LIN {X 0,Y 168.066,Z 1160.336,A -85,B 0,C 180,E1 3860.949,E2 3860.949} C_VEL
LIN {X 0,Y 168.839,Z 1157.716,A -85,B 0,C 180,E1 3853.839,E2 3853.839} C_VEL
LIN {X 0,Y 170.872,Z 1154.031,A -85,B 0,C 180,E1 3847.282,E2 3847.282} C_VEL
LIN {X 0,Y 175.431,Z 1147.884,A -85,B 0,C 180,E1 3839.519,E2 3839.519} C_VEL
LIN {X 0,Y 182.099,Z 1140.235,A -85,B 0,C 180,E1 3832.449,E2 3832.449} C_VEL
LIN {X 0,Y 190.542,Z 1131.041,A -85,B 0,C 180,E1 3826.159,E2 3826.159} C_VEL
LIN {X 0,Y 200.886,Z 1120.046,A -85,B 0,C 180,E1 3820.401,E2 3820.401} C_VEL
LIN {X 0,Y 211.702,Z 1108.233,A -85,B 0,C 180,E1 3815.674,E2 3815.674} C_VEL
LIN {X 0,Y 223.761,Z 1094.432,A -85,B 0,C 180,E1 3811.409,E2 3811.409} C_VEL
LIN {X 0,Y 235.465,Z 1080.228,A -85,B 0,C 180,E1 3807.965,E2 3807.965} C_VEL
LIN {X 0,Y 247.528,Z 1064.175,A -85,B 0,C 180,E1 3804.927,E2 3804.927} C_VEL
LIN {X 0,Y 259.432,Z 1046.898,A -85,B 0,C 180,E1 3802.336,E2 3802.336} C_VEL
LIN {X 0,Y 270.34,Z 1029.197,A -85,B 0,C 180,E1 3800.24,E2 3800.24} C_VEL
LIN {X 0,Y 281.272,Z 1009.124,A -85,B 0,C 180,E1 3798.354,E2 3798.354} C_VEL
LIN {X 0,Y 290.529,Z 989.805,A -85,B 0,C 180,E1 3796.914,E2 3796.914} C_VEL
LIN {X 0,Y 299.081,Z 968.565,A -85,B 0,C 180,E1 3795.673,E2 3795.673} C_VEL
LIN {X 0,Y 306.639,Z 946.026,A -85,B 0,C 180,E1 3794.652,E2 3794.652} C_VEL
LIN {X 0,Y 312.105,Z 925.795,A -85,B 0,C 180,E1 3793.953,E2 3793.953} C_VEL
LIN {X 0,Y 316.755,Z 902.819,A -85,B 0,C 180,E1 3793.358,E2 3793.358} C_VEL
LIN {X 0,Y 319.982,Z 878.763,A -85,B 0,C 180,E1 3792.859,E2 3792.859} C_VEL
LIN {X 0,Y 334.332,Z 738.673,A -85,B 0,C 180,E1 3790.249,E2 3790.249} C_VEL
LIN {X 0,Y 331.548,Z 732.932,A -85,B 0,C 180,E1 3787.189,E2 3787.189} C_VEL
LIN {X 0,Y 329.463,Z 728.967,A -85,B 0,C 180,E1 3784.002,E2 3784.002} C_VEL
LIN {X 0,Y 327.825,Z 726.055,A -85,B 0,C 180,E1 3778.951,E2 3778.951} C_VEL
LIN {X 0,Y 327.708,Z 726.631,A -85,B 0,C 180,E1 3776.501,E2 3776.501} C_VEL
LIN {X 0,Y 328.643,Z 729.356,A -85,B 0,C 180,E1 3772.394,E2 3772.394} C_VEL
LIN {X 0,Y 330.208,Z 733.352,A -85,B 0,C 180,E1 3769.356,E2 3769.356} C_VEL
LIN {X 0,Y 332.385,Z 738.672,A -85,B 0,C 180,E1 3766.474,E2 3766.474} C_VEL
LIN {X 0,Y 333.349,Z 741.398,A -85,B 0,C 180,E1 3765.384,E2 3765.384} C_VEL
LIN {X 0,Y 317.82,Z 895.127,A -85,B 0,C 180,E1 3762.622,E2 3762.622} C_VEL
LIN {X 0,Y 313.848,Z 917.711,A -85,B 0,C 180,E1 3762.113,E2 3762.113} C_VEL
LIN {X 0,Y 308.482,Z 939.763,A -85,B 0,C 180,E1 3761.453,E2 3761.453} C_VEL
LIN {X 0,Y 302.074,Z 960.282,A -85,B 0,C 180,E1 3760.622,E2 3760.622} C_VEL
LIN {X 0,Y 294.064,Z 981.25,A -85,B 0,C 180,E1 3759.511,E2 3759.511} C_VEL
LIN {X 0,Y 285.141,Z 1001.061,A -85,B 0,C 180,E1 3758.179,E2 3758.179} C_VEL
LIN {X 0,Y 275.576,Z 1019.159,A -85,B 0,C 180,E1 3756.628,E2 3756.628} C_VEL
LIN {X 0,Y 263.972,Z 1038.466,A -85,B 0,C 180,E1 3754.538,E2 3754.538} C_VEL
LIN {X 0,Y 252.604,Z 1055.305,A -85,B 0,C 180,E1 3752.21,E2 3752.21} C_VEL
LIN {X 0,Y 240.489,Z 1071.192,A -85,B 0,C 180,E1 3749.387,E2 3749.387} C_VEL
LIN {X 0,Y 228.005,Z 1086.134,A -85,B 0,C 180,E1 3745.977,E2 3745.977} C_VEL
LIN {X 0,Y 215.781,Z 1099.645,A -85,B 0,C 180,E1 3741.973,E2 3741.973} C_VEL
LIN {X 0,Y 204.128,Z 1111.522,A -85,B 0,C 180,E1 3737.285,E2 3737.285} C_VEL
LIN {X 0,Y 193.43,Z 1121.957,A -85,B 0,C 180,E1 3731.822,E2 3731.822} C_VEL
LIN {X 0,Y 184.531,Z 1130.557,A -85,B 0,C 180,E1 3725.816,E2 3725.816} C_VEL
LIN {X 0,Y 177.286,Z 1137.575,A -85,B 0,C 180,E1 3719.014,E2 3719.014} C_VEL
LIN {X 0,Y 172.1,Z 1143.09,A -85,B 0,C 180,E1 3711.47,E2 3711.47} C_VEL
LIN {X 0,Y 169.41,Z 1146.62,A -85,B 0,C 180,E1 3704.352,E2 3704.352} C_VEL
LIN {X 0,Y 168.309,Z 1148.543,A -85,B 0,C 180,E1 3697.51,E2 3697.51} C_VEL
LIN {X 0,Y 168.074,Z 1149.252,A -85,B 0,C 180,E1 3691.704,E2 3691.704} C_VEL
LIN {X 0,Y 168.13,Z 1149.097,A -85,B 0,C 180,E1 3685.566,E2 3685.566} C_VEL
LIN {X 0,Y 168.751,Z 1147.654,A -85,B 0,C 180,E1 3678.724,E2 3678.724} C_VEL
LIN {X 0,Y 170.661,Z 1144.912,A -85,B 0,C 180,E1 3671.646,E2 3671.646} C_VEL
LIN {X 0,Y 174.681,Z 1140.291,A -85,B 0,C 180,E1 3664.213,E2 3664.213} C_VEL
LIN {X 0,Y 180.983,Z 1133.995,A -85,B 0,C 180,E1 3657.114,E2 3657.114} C_VEL
LIN {X 0,Y 188.87,Z 1126.429,A -85,B 0,C 180,E1 3650.951,E2 3650.951} C_VEL
LIN {X 0,Y 198.846,Z 1116.798,A -85,B 0,C 180,E1 3645.154,E2 3645.154} C_VEL
LIN {X 0,Y 209.674,Z 1106.072,A -85,B 0,C 180,E1 3640.272,E2 3640.272} C_VEL
LIN {X 0,Y 221.323,Z 1093.753,A -85,B 0,C 180,E1 3636.035,E2 3636.035} C_VEL
LIN {X 0,Y 231.633,Z 1082.102,A -85,B 0,C 180,E1 3632.876,E2 3632.876} C_VEL
LIN {X 0,Y 216.361,Z 1086.384,A -85,B 0,C 180,E1 3628.424,E2 3628.424} C_VEL
LIN {X 0,Y 206.073,Z 1089.051,A -85,B 0,C 180,E1 3624.358,E2 3624.358} C_VEL
LIN {X 0,Y 199.167,Z 1090.87,A -85,B 0,C 180,E1 3620.882,E2 3620.882} C_VEL
LIN {X 0,Y 192.703,Z 1092.575,A -85,B 0,C 180,E1 3616.582,E2 3616.582} C_VEL
LIN {X 0,Y 187.91,Z 1093.996,A -85,B 0,C 180,E1 3612.289,E2 3612.289} C_VEL
LIN {X 0,Y 184.075,Z 1095.335,A -85,B 0,C 180,E1 3607.178,E2 3607.178} C_VEL
LIN {X 0,Y 181.631,Z 1096.889,A -85,B 0,C 180,E1 3600.316,E2 3600.316} C_VEL
LIN {X 0,Y 183.368,Z 1099.077,A -85,B 0,C 180,E1 3589.635,E2 3589.635} C_VEL
LIN {X 0,Y 190.031,Z 1099.894,A -85,B 0,C 180,E1 3581.916,E2 3581.916} C_VEL
LIN {X 0,Y 196.11,Z 1100.057,A -85,B 0,C 180,E1 3577.582,E2 3577.582} C_VEL
LIN {X 0,Y 199.24,Z 1100.523,A -85,B 0,C 180,E1 3575.354,E2 3575.354} C_VEL
LIN {X 0,Y 205.611,Z 1103.158,A -85,B 0,C 180,E1 3570.193,E2 3570.193} C_VEL
LIN {X 0,Y 209.729,Z 1103.302,A -85,B 0,C 180,E1 3568.398,E2 3568.398} C_VEL
LIN {X 0,Y 211.44,Z 1103.162,A -85,B 0,C 180,E1 3567.829,E2 3567.829} C_VEL
LIN {X 0,Y 198.52,Z 1116.738,A -85,B 0,C 180,E1 3562.816,E2 3562.816} C_VEL
LIN {X 0,Y 187.536,Z 1127.926,A -85,B 0,C 180,E1 3557.372,E2 3557.372} C_VEL
LIN {X 0,Y 177.906,Z 1137.495,A -85,B 0,C 180,E1 3551.114,E2 3551.114} C_VEL
LIN {X 0,Y 169.726,Z 1146.03,A -85,B 0,C 180,E1 3543.625,E2 3543.625} C_VEL
LIN {X 0,Y 164.54,Z 1152.122,A -85,B 0,C 180,E1 3536.334,E2 3536.334} C_VEL
LIN {X 0,Y 161.344,Z 1156.757,A -85,B 0,C 180,E1 3528.424,E2 3528.424} C_VEL
LIN {X 0,Y 160.19,Z 1159.484,A -85,B 0,C 180,E1 3521.499,E2 3521.499} C_VEL
LIN {X 0,Y 160.016,Z 1160.978,A -85,B 0,C 180,E1 3514.659,E2 3514.659} C_VEL
LIN {X 0,Y 160.047,Z 1161.226,A -85,B 0,C 180,E1 3508.926,E2 3508.926} C_VEL
LIN {X 0,Y 160.011,Z 1160.594,A -85,B 0,C 180,E1 3503.181,E2 3503.181} C_VEL
LIN {X 0,Y 160.338,Z 1158.972,A -85,B 0,C 180,E1 3497.027,E2 3497.027} C_VEL
LIN {X 0,Y 162.006,Z 1155.698,A -85,B 0,C 180,E1 3489.403,E2 3489.403} C_VEL
LIN {X 0,Y 165.624,Z 1150.678,A -85,B 0,C 180,E1 3481.808,E2 3481.808} C_VEL
LIN {X 0,Y 171.617,Z 1143.989,A -85,B 0,C 180,E1 3474.366,E2 3474.366} C_VEL
LIN {X 0,Y 179.581,Z 1135.749,A -85,B 0,C 180,E1 3467.647,E2 3467.647} C_VEL
LIN {X 0,Y 190.084,Z 1125.198,A -85,B 0,C 180,E1 3461.219,E2 3461.219} C_VEL
LIN {X 0,Y 201.378,Z 1113.79,A -85,B 0,C 180,E1 3455.971,E2 3455.971} C_VEL
LIN {X 0,Y 213.404,Z 1100.89,A -85,B 0,C 180,E1 3451.491,E2 3451.491} C_VEL
LIN {X 0,Y 226.562,Z 1085.934,A -85,B 0,C 180,E1 3447.495,E2 3447.495} C_VEL
LIN {X 0,Y 239.155,Z 1070.454,A -85,B 0,C 180,E1 3444.298,E2 3444.298} C_VEL
LIN {X 0,Y 251.201,Z 1054.032,A -85,B 0,C 180,E1 3441.657,E2 3441.657} C_VEL
LIN {X 0,Y 262.913,Z 1036.48,A -85,B 0,C 180,E1 3439.412,E2 3439.412} C_VEL
LIN {X 0,Y 273.298,Z 1018.853,A -85,B 0,C 180,E1 3437.628,E2 3437.628} C_VEL
LIN {X 0,Y 283.934,Z 998.39,A -85,B 0,C 180,E1 3435.98,E2 3435.98} C_VEL
LIN {X 0,Y 292.6,Z 979.055,A -85,B 0,C 180,E1 3434.748,E2 3434.748} C_VEL
LIN {X 0,Y 300.502,Z 958.071,A -85,B 0,C 180,E1 3433.694,E2 3433.694} C_VEL
LIN {X 0,Y 307.329,Z 936.133,A -85,B 0,C 180,E1 3432.838,E2 3432.838} C_VEL
LIN {X 0,Y 312.656,Z 913.731,A -85,B 0,C 180,E1 3432.199,E2 3432.199} C_VEL
LIN {X 0,Y 316.677,Z 889.714,A -85,B 0,C 180,E1 3431.675,E2 3431.675} C_VEL
LIN {X 0,Y 332.049,Z 744.44,A -85,B 0,C 180,E1 3429.008,E2 3429.008} C_VEL
LIN {X 0,Y 329.883,Z 739.96,A -85,B 0,C 180,E1 3426.351,E2 3426.351} C_VEL
LIN {X 0,Y 328.38,Z 736.839,A -85,B 0,C 180,E1 3423.84,E2 3423.84} C_VEL
LIN {X 0,Y 326.831,Z 733.964,A -85,B 0,C 180,E1 3418.772,E2 3418.772} C_VEL
LIN {X 0,Y 326.748,Z 734.814,A -85,B 0,C 180,E1 3416.139,E2 3416.139} C_VEL
LIN {X 0,Y 327.589,Z 737.286,A -85,B 0,C 180,E1 3412.546,E2 3412.546} C_VEL
LIN {X 0,Y 329.057,Z 741.202,A -85,B 0,C 180,E1 3409.584,E2 3409.584} C_VEL
LIN {X 0,Y 331.095,Z 746.453,A -85,B 0,C 180,E1 3406.776,E2 3406.776} C_VEL
LIN {X 0,Y 331.165,Z 747.084,A -85,B 0,C 180,E1 3406.642,E2 3406.642} C_VEL
LIN {X 0,Y 315.809,Z 895.146,A -85,B 0,C 180,E1 3404.026,E2 3404.026} C_VEL
LIN {X 0,Y 311.75,Z 917.772,A -85,B 0,C 180,E1 3403.53,E2 3403.53} C_VEL
LIN {X 0,Y 306.264,Z 939.882,A -85,B 0,C 180,E1 3402.891,E2 3402.891} C_VEL
LIN {X 0,Y 299.957,Z 959.745,A -85,B 0,C 180,E1 3402.115,E2 3402.115} C_VEL
LIN {X 0,Y 291.791,Z 980.838,A -85,B 0,C 180,E1 3401.041,E2 3401.041} C_VEL
LIN {X 0,Y 282.894,Z 1000.319,A -85,B 0,C 180,E1 3399.782,E2 3399.782} C_VEL
LIN {X 0,Y 272.487,Z 1019.611,A -85,B 0,C 180,E1 3398.18,E2 3398.18} C_VEL
LIN {X 0,Y 260.713,Z 1038.7,A -85,B 0,C 180,E1 3396.159,E2 3396.159} C_VEL
LIN {X 0,Y 248.93,Z 1055.677,A -85,B 0,C 180,E1 3393.86,E2 3393.86} C_VEL
LIN {X 0,Y 236.455,Z 1071.542,A -85,B 0,C 180,E1 3391.082,E2 3391.082} C_VEL
LIN {X 0,Y 223.549,Z 1086.464,A -85,B 0,C 180,E1 3387.708,E2 3387.708} C_VEL
LIN {X 0,Y 211.489,Z 1099.298,A -85,B 0,C 180,E1 3383.944,E2 3383.944} C_VEL
LIN {X 0,Y 199.818,Z 1110.717,A -85,B 0,C 180,E1 3379.516,E2 3379.516} C_VEL
LIN {X 0,Y 188.909,Z 1120.93,A -85,B 0,C 180,E1 3374.319,E2 3374.319} C_VEL
LIN {X 0,Y 179.601,Z 1129.317,A -85,B 0,C 180,E1 3368.574,E2 3368.574} C_VEL
LIN {X 0,Y 171.32,Z 1136.805,A -85,B 0,C 180,E1 3361.559,E2 3361.559} C_VEL
LIN {X 0,Y 165.538,Z 1142.429,A -85,B 0,C 180,E1 3354.208,E2 3354.208} C_VEL
LIN {X 0,Y 162.098,Z 1146.161,A -85,B 0,C 180,E1 3346.852,E2 3346.852} C_VEL
LIN {X 0,Y 160.483,Z 1148.584,A -85,B 0,C 180,E1 3339.322,E2 3339.322} C_VEL
LIN {X 0,Y 160.089,Z 1149.48,A -85,B 0,C 180,E1 3332.864,E2 3332.864} C_VEL
LIN {X 0,Y 160.085,Z 1149.51,A -85,B 0,C 180,E1 3327.494,E2 3327.494} C_VEL
LIN {X 0,Y 160.396,Z 1148.736,A -85,B 0,C 180,E1 3321.396,E2 3321.396} C_VEL
LIN {X 0,Y 161.958,Z 1146.373,A -85,B 0,C 180,E1 3313.502,E2 3313.502} C_VEL
LIN {X 0,Y 165.444,Z 1142.551,A -85,B 0,C 180,E1 3305.865,E2 3305.865} C_VEL
LIN {X 0,Y 171.142,Z 1137.021,A -85,B 0,C 180,E1 3298.538,E2 3298.538} C_VEL
LIN {X 0,Y 179.099,Z 1129.86,A -85,B 0,C 180,E1 3291.707,E2 3291.707} C_VEL
LIN {X 0,Y 188.81,Z 1121.095,A -85,B 0,C 180,E1 3285.651,E2 3285.651} C_VEL
LIN {X 0,Y 199.71,Z 1110.923,A -85,B 0,C 180,E1 3280.448,E2 3280.448} C_VEL
LIN {X 0,Y 211.376,Z 1099.547,A -85,B 0,C 180,E1 3276.014,E2 3276.014} C_VEL
LIN {X 0,Y 221.91,Z 1088.357,A -85,B 0,C 180,E1 3272.654,E2 3272.654} C_VEL
LIN {X 0,Y 211.435,Z 1091.167,A -85,B 0,C 180,E1 3269.527,E2 3269.527} C_VEL
LIN {X 0,Y 201.236,Z 1093.692,A -85,B 0,C 180,E1 3265.612,E2 3265.612} C_VEL
LIN {X 0,Y 193.118,Z 1095.612,A -85,B 0,C 180,E1 3261.568,E2 3261.568} C_VEL
LIN {X 0,Y 187.13,Z 1097.099,A -85,B 0,C 180,E1 3257.732,E2 3257.732} C_VEL
LIN {X 0,Y 181.506,Z 1098.586,A -85,B 0,C 180,E1 3252.73,E2 3252.73} C_VEL
LIN {X 0,Y 177.713,Z 1099.879,A -85,B 0,C 180,E1 3247.761,E2 3247.761} C_VEL
LIN {X 0,Y 175.075,Z 1101.482,A -85,B 0,C 180,E1 3240.328,E2 3240.328} C_VEL
LIN {X 0,Y 176.758,Z 1103.63,A -85,B 0,C 180,E1 3229.572,E2 3229.572} C_VEL
LIN {X 0,Y 183.457,Z 1104.491,A -85,B 0,C 180,E1 3221.573,E2 3221.573} C_VEL
LIN {X 0,Y 191.592,Z 1104.607,A -85,B 0,C 180,E1 3215.981,E2 3215.981} C_VEL
LIN {X 0,Y 203.409,Z 1103.964,A -85,B 0,C 180,E1 3210.558,E2 3210.558} C_VEL
LIN {X 0,Y 209.729,Z 1103.302,A -85,B 0,C 180,E1 3208.398,E2 3208.398} C_VEL
LIN {X 0,Y 210.064,Z 1103.848,A -85,B 0,C 180,E1 3207.907,E2 3207.907} C_VEL
LIN {X 0,Y 208.692,Z 1105.572,A -85,B 0,C 180,E1 3207.279,E2 3207.279} C_VEL
LIN {X 0,Y 205.22,Z 1108.258,A -85,B 0,C 180,E1 3206.659,E2 3206.659} C_VEL
LIN {X 0,Y 196.789,Z 1113.88,A -85,B 0,C 180,E1 3205.674,E2 3205.674} C_VEL
LIN {X 0,Y 193.755,Z 1116.236,A -85,B 0,C 180,E1 3204.876,E2 3204.876} C_VEL
LIN {X 0,Y 181.945,Z 1127.613,A -85,B 0,C 180,E1 3199.321,E2 3199.321} C_VEL
LIN {X 0,Y 171.674,Z 1137.184,A -85,B 0,C 180,E1 3192.956,E2 3192.956} C_VEL
LIN {X 0,Y 162.826,Z 1145.732,A -85,B 0,C 180,E1 3185.246,E2 3185.246} C_VEL
LIN {X 0,Y 157.136,Z 1151.819,A -85,B 0,C 180,E1 3177.678,E2 3177.678} C_VEL
LIN {X 0,Y 153.574,Z 1156.459,A -85,B 0,C 180,E1 3169.393,E2 3169.393} C_VEL
LIN {X 0,Y 152.246,Z 1159.182,A -85,B 0,C 180,E1 3162.132,E2 3162.132} C_VEL
LIN {X 0,Y 152.013,Z 1160.659,A -85,B 0,C 180,E1 3155.284,E2 3155.284} C_VEL
LIN {X 0,Y 152.05,Z 1160.959,A -85,B 0,C 180,E1 3149.247,E2 3149.247} C_VEL
LIN {X 0,Y 152.014,Z 1160.375,A -85,B 0,C 180,E1 3143.201,E2 3143.201} C_VEL
LIN {X 0,Y 152.366,Z 1158.799,A -85,B 0,C 180,E1 3136.722,E2 3136.722} C_VEL
LIN {X 0,Y 154.054,Z 1155.753,A -85,B 0,C 180,E1 3129.086,E2 3129.086} C_VEL
LIN {X 0,Y 158.043,Z 1150.711,A -85,B 0,C 180,E1 3120.847,E2 3120.847} C_VEL
LIN {X 0,Y 164.538,Z 1144.048,A -85,B 0,C 180,E1 3113.015,E2 3113.015} C_VEL
LIN {X 0,Y 173.013,Z 1135.859,A -85,B 0,C 180,E1 3106.093,E2 3106.093} C_VEL
LIN {X 0,Y 184.457,Z 1125.072,A -85,B 0,C 180,E1 3099.36,E2 3099.36} C_VEL
LIN {X 0,Y 196.558,Z 1113.462,A -85,B 0,C 180,E1 3093.988,E2 3093.988} C_VEL
LIN {X 0,Y 209.352,Z 1100.343,A -85,B 0,C 180,E1 3089.466,E2 3089.466} C_VEL
LIN {X 0,Y 223.373,Z 1084.955,A -85,B 0,C 180,E1 3085.449,E2 3085.449} C_VEL
LIN {X 0,Y 236.638,Z 1069.116,A -85,B 0,C 180,E1 3082.281,E2 3082.281} C_VEL
LIN {X 0,Y 249.192,Z 1052.348,A -85,B 0,C 180,E1 3079.696,E2 3079.696} C_VEL
LIN {X 0,Y 261.961,Z 1033.33,A -85,B 0,C 180,E1 3077.406,E2 3077.406} C_VEL
LIN {X 0,Y 273.075,Z 1014.66,A -85,B 0,C 180,E1 3075.641,E2 3075.641} C_VEL
LIN {X 0,Y 283.102,Z 995.111,A -85,B 0,C 180,E1 3074.192,E2 3074.192} C_VEL
LIN {X 0,Y 291.964,Z 975.24,A -85,B 0,C 180,E1 3073.018,E2 3073.018} C_VEL
LIN {X 0,Y 299.128,Z 956.022,A -85,B 0,C 180,E1 3072.12,E2 3072.12} C_VEL
LIN {X 0,Y 306.111,Z 933.229,A -85,B 0,C 180,E1 3071.294,E2 3071.294} C_VEL
LIN {X 0,Y 311.322,Z 911.208,A -85,B 0,C 180,E1 3070.707,E2 3070.707} C_VEL
LIN {X 0,Y 315.043,Z 888.222,A -85,B 0,C 180,E1 3070.228,E2 3070.228} C_VEL
LIN {X 0,Y 329.913,Z 750.378,A -85,B 0,C 180,E1 3067.75,E2 3067.75} C_VEL
LIN {X 0,Y 328.35,Z 747.083,A -85,B 0,C 180,E1 3065.591,E2 3065.591} C_VEL
LIN {X 0,Y 327.21,Z 744.588,A -85,B 0,C 180,E1 3063.503,E2 3063.503} C_VEL
LIN {X 0,Y 325.856,Z 741.909,A -85,B 0,C 180,E1 3058.769,E2 3058.769} C_VEL
LIN {X 0,Y 325.759,Z 742.699,A -85,B 0,C 180,E1 3056.304,E2 3056.304} C_VEL
LIN {X 0,Y 326.514,Z 745.1,A -85,B 0,C 180,E1 3052.787,E2 3052.787} C_VEL
LIN {X 0,Y 327.861,Z 748.907,A -85,B 0,C 180,E1 3049.9,E2 3049.9} C_VEL
LIN {X 0,Y 329.155,Z 752.529,A -85,B 0,C 180,E1 3047.92,E2 3047.92} C_VEL
LIN {X 0,Y 314.011,Z 894.992,A -85,B 0,C 180,E1 3045.451,E2 3045.451} C_VEL
LIN {X 0,Y 309.874,Z 917.703,A -85,B 0,C 180,E1 3044.969,E2 3044.969} C_VEL
LIN {X 0,Y 304.241,Z 940,A -85,B 0,C 180,E1 3044.349,E2 3044.349} C_VEL
LIN {X 0,Y 297.606,Z 960.483,A -85,B 0,C 180,E1 3043.575,E2 3043.575} C_VEL
LIN {X 0,Y 289.293,Z 981.419,A -85,B 0,C 180,E1 3042.539,E2 3042.539} C_VEL
LIN {X 0,Y 280.225,Z 1000.82,A -85,B 0,C 180,E1 3041.32,E2 3041.32} C_VEL
LIN {X 0,Y 270.066,Z 1019.262,A -85,B 0,C 180,E1 3039.837,E2 3039.837} C_VEL
LIN {X 0,Y 257.968,Z 1038.499,A -85,B 0,C 180,E1 3037.872,E2 3037.872} C_VEL
LIN {X 0,Y 245.867,Z 1055.521,A -85,B 0,C 180,E1 3035.635,E2 3035.635} C_VEL
LIN {X 0,Y 233.245,Z 1071.161,A -85,B 0,C 180,E1 3032.973,E2 3032.973} C_VEL
LIN {X 0,Y 220.026,Z 1086.037,A -85,B 0,C 180,E1 3029.702,E2 3029.702} C_VEL
LIN {X 0,Y 207.46,Z 1098.936,A -85,B 0,C 180,E1 3025.992,E2 3025.992} C_VEL
LIN {X 0,Y 195.214,Z 1110.471,A -85,B 0,C 180,E1 3021.596,E2 3021.596} C_VEL
LIN {X 0,Y 183.676,Z 1120.789,A -85,B 0,C 180,E1 3016.386,E2 3016.386} C_VEL
LIN {X 0,Y 173.268,Z 1129.62,A -85,B 0,C 180,E1 3010.264,E2 3010.264} C_VEL
LIN {X 0,Y 164.511,Z 1137.013,A -85,B 0,C 180,E1 3003.161,E2 3003.161} C_VEL
LIN {X 0,Y 158.158,Z 1142.704,A -85,B 0,C 180,E1 2995.461,E2 2995.461} C_VEL
LIN {X 0,Y 154.349,Z 1146.456,A -85,B 0,C 180,E1 2987.726,E2 2987.726} C_VEL
LIN {X 0,Y 152.548,Z 1148.877,A -85,B 0,C 180,E1 2979.812,E2 2979.812} C_VEL
LIN {X 0,Y 152.097,Z 1149.771,A -85,B 0,C 180,E1 2973.015,E2 2973.015} C_VEL
LIN {X 0,Y 152.091,Z 1149.801,A -85,B 0,C 180,E1 2967.362,E2 2967.362} C_VEL
LIN {X 0,Y 152.443,Z 1149.028,A -85,B 0,C 180,E1 2960.943,E2 2960.943} C_VEL
LIN {X 0,Y 154.196,Z 1146.668,A -85,B 0,C 180,E1 2952.646,E2 2952.646} C_VEL
LIN {X 0,Y 157.881,Z 1142.976,A -85,B 0,C 180,E1 2944.893,E2 2944.893} C_VEL
LIN {X 0,Y 164.098,Z 1137.416,A -85,B 0,C 180,E1 2937.161,E2 2937.161} C_VEL
LIN {X 0,Y 172.737,Z 1130.161,A -85,B 0,C 180,E1 2930.021,E2 2930.021} C_VEL
LIN {X 0,Y 182.708,Z 1121.67,A -85,B 0,C 180,E1 2924.028,E2 2924.028} C_VEL
LIN {X 0,Y 194.497,Z 1111.231,A -85,B 0,C 180,E1 2918.611,E2 2918.611} C_VEL
LIN {X 0,Y 206.99,Z 1099.549,A -85,B 0,C 180,E1 2914.08,E2 2914.08} C_VEL
LIN {X 0,Y 211.969,Z 1094.464,A -85,B 0,C 180,E1 2912.45,E2 2912.45} C_VEL
LIN {X 0,Y 196.359,Z 1098.097,A -85,B 0,C 180,E1 2906.949,E2 2906.949} C_VEL
LIN {X 0,Y 183.195,Z 1101.206,A -85,B 0,C 180,E1 2900.112,E2 2900.112} C_VEL
LIN {X 0,Y 171.637,Z 1104.182,A -85,B 0,C 180,E1 2889.05,E2 2889.05} C_VEL
LIN {X 0,Y 169.799,Z 1107.852,A -85,B 0,C 180,E1 2869.826,E2 2869.826} C_VEL
LIN {X 0,Y 176.708,Z 1108.791,A -85,B 0,C 180,E1 2861.186,E2 2861.186} C_VEL
LIN {X 0,Y 185.45,Z 1108.965,A -85,B 0,C 180,E1 2855.132,E2 2855.132} C_VEL
LIN {X 0,Y 197.588,Z 1108.421,A -85,B 0,C 180,E1 2849.601,E2 2849.601} C_VEL
LIN {X 0,Y 202.008,Z 1108.039,A -85,B 0,C 180,E1 2848.064,E2 2848.064} C_VEL
LIN {X 0,Y 193.755,Z 1116.236,A -85,B 0,C 180,E1 2844.876,E2 2844.876} C_VEL
LIN {X 0,Y 189.106,Z 1120.152,A -85,B 0,C 180,E1 2843.4,E2 2843.4} C_VEL
LIN {X 0,Y 174.971,Z 1129.302,A -85,B 0,C 180,E1 2839.934,E2 2839.934} C_VEL
LIN {X 0,Y 170.613,Z 1132.534,A -85,B 0,C 180,E1 2838.109,E2 2838.109} C_VEL
LIN {X 0,Y 160.546,Z 1141.375,A -85,B 0,C 180,E1 2831.101,E2 2831.101} C_VEL
LIN {X 0,Y 152.816,Z 1148.567,A -85,B 0,C 180,E1 2823.34,E2 2823.34} C_VEL
LIN {X 0,Y 147.706,Z 1153.814,A -85,B 0,C 180,E1 2815.244,E2 2815.244} C_VEL
LIN {X 0,Y 144.832,Z 1157.781,A -85,B 0,C 180,E1 2806.442,E2 2806.442} C_VEL
LIN {X 0,Y 144.065,Z 1159.796,A -85,B 0,C 180,E1 2798.783,E2 2798.783} C_VEL
LIN {X 0,Y 144.036,Z 1160.549,A -85,B 0,C 180,E1 2792.785,E2 2792.785} C_VEL
LIN {X 0,Y 144.043,Z 1160.571,A -85,B 0,C 180,E1 2787.613,E2 2787.613} C_VEL
LIN {X 0,Y 144.049,Z 1159.86,A -85,B 0,C 180,E1 2781.619,E2 2781.619} C_VEL
LIN {X 0,Y 144.685,Z 1158.011,A -85,B 0,C 180,E1 2774.365,E2 2774.365} C_VEL
LIN {X 0,Y 147.338,Z 1154.222,A -85,B 0,C 180,E1 2765.546,E2 2765.546} C_VEL
LIN {X 0,Y 152.222,Z 1149.065,A -85,B 0,C 180,E1 2757.411,E2 2757.411} C_VEL
LIN {X 0,Y 159.901,Z 1141.895,A -85,B 0,C 180,E1 2749.435,E2 2749.435} C_VEL
LIN {X 0,Y 169.566,Z 1133.424,A -85,B 0,C 180,E1 2742.517,E2 2742.517} C_VEL
LIN {X 0,Y 181.247,Z 1122.963,A -85,B 0,C 180,E1 2736.349,E2 2736.349} C_VEL
LIN {X 0,Y 194.798,Z 1110.385,A -85,B 0,C 180,E1 2730.881,E2 2730.881} C_VEL
LIN {X 0,Y 208.068,Z 1097.345,A -85,B 0,C 180,E1 2726.643,E2 2726.643} C_VEL
LIN {X 0,Y 221.674,Z 1082.643,A -85,B 0,C 180,E1 2723.053,E2 2723.053} C_VEL
LIN {X 0,Y 236.039,Z 1065.64,A -85,B 0,C 180,E1 2719.882,E2 2719.882} C_VEL
LIN {X 0,Y 248.926,Z 1048.73,A -85,B 0,C 180,E1 2717.452,E2 2717.452} C_VEL
LIN {X 0,Y 260.999,Z 1030.713,A -85,B 0,C 180,E1 2715.445,E2 2715.445} C_VEL
LIN {X 0,Y 272.733,Z 1010.921,A -85,B 0,C 180,E1 2713.708,E2 2713.708} C_VEL
LIN {X 0,Y 282.549,Z 991.834,A -85,B 0,C 180,E1 2712.396,E2 2712.396} C_VEL
LIN {X 0,Y 291.658,Z 970.97,A -85,B 0,C 180,E1 2711.268,E2 2711.268} C_VEL
LIN {X 0,Y 299.269,Z 950.317,A -85,B 0,C 180,E1 2710.393,E2 2710.393} C_VEL
LIN {X 0,Y 305.458,Z 929.062,A -85,B 0,C 180,E1 2709.708,E2 2709.708} C_VEL
LIN {X 0,Y 310.715,Z 905.521,A -85,B 0,C 180,E1 2709.14,E2 2709.14} C_VEL
LIN {X 0,Y 314.102,Z 882.99,A -85,B 0,C 180,E1 2708.699,E2 2708.699} C_VEL
LIN {X 0,Y 327.933,Z 756.407,A -85,B 0,C 180,E1 2706.477,E2 2706.477} C_VEL
LIN {X 0,Y 326.135,Z 752.46,A -85,B 0,C 180,E1 2703.339,E2 2703.339} C_VEL
LIN {X 0,Y 324.865,Z 749.822,A -85,B 0,C 180,E1 2698.589,E2 2698.589} C_VEL
LIN {X 0,Y 324.864,Z 751.206,A -85,B 0,C 180,E1 2695.41,E2 2695.41} C_VEL
LIN {X 0,Y 325.474,Z 753.027,A -85,B 0,C 180,E1 2692.941,E2 2692.941} C_VEL
LIN {X 0,Y 326.67,Z 756.596,A -85,B 0,C 180,E1 2690.228,E2 2690.228} C_VEL
LIN {X 0,Y 327.249,Z 758.491,A -85,B 0,C 180,E1 2689.203,E2 2689.203} C_VEL
LIN {X 0,Y 312.385,Z 895.027,A -85,B 0,C 180,E1 2686.887,E2 2686.887} C_VEL
LIN {X 0,Y 308.194,Z 917.626,A -85,B 0,C 180,E1 2686.425,E2 2686.425} C_VEL
LIN {X 0,Y 302.423,Z 940.102,A -85,B 0,C 180,E1 2685.825,E2 2685.825} C_VEL
LIN {X 0,Y 295.452,Z 961.218,A -85,B 0,C 180,E1 2685.057,E2 2685.057} C_VEL
LIN {X 0,Y 286.997,Z 982.001,A -85,B 0,C 180,E1 2684.061,E2 2684.061} C_VEL
LIN {X 0,Y 277.323,Z 1002.107,A -85,B 0,C 180,E1 2682.83,E2 2682.83} C_VEL
LIN {X 0,Y 266.93,Z 1020.508,A -85,B 0,C 180,E1 2681.385,E2 2681.385} C_VEL
LIN {X 0,Y 254.619,Z 1039.493,A -85,B 0,C 180,E1 2679.482,E2 2679.482} C_VEL
LIN {X 0,Y 242.228,Z 1056.408,A -85,B 0,C 180,E1 2677.3,E2 2677.3} C_VEL
LIN {X 0,Y 229.041,Z 1072.241,A -85,B 0,C 180,E1 2674.641,E2 2674.641} C_VEL
LIN {X 0,Y 215.285,Z 1087.12,A -85,B 0,C 180,E1 2671.376,E2 2671.376} C_VEL
LIN {X 0,Y 202.31,Z 1099.945,A -85,B 0,C 180,E1 2667.685,E2 2667.685} C_VEL
LIN {X 0,Y 189.599,Z 1111.341,A -85,B 0,C 180,E1 2663.282,E2 2663.282} C_VEL
LIN {X 0,Y 176.989,Z 1121.983,A -85,B 0,C 180,E1 2657.736,E2 2657.736} C_VEL
LIN {X 0,Y 166.151,Z 1130.708,A -85,B 0,C 180,E1 2651.449,E2 2651.449} C_VEL
LIN {X 0,Y 157.031,Z 1137.858,A -85,B 0,C 180,E1 2644.13,E2 2644.13} C_VEL
LIN {X 0,Y 150.086,Z 1143.588,A -85,B 0,C 180,E1 2635.66,E2 2635.66} C_VEL
LIN {X 0,Y 146.227,Z 1147.205,A -85,B 0,C 180,E1 2627.509,E2 2627.509} C_VEL
LIN {X 0,Y 144.464,Z 1149.357,A -85,B 0,C 180,E1 2619.16,E2 2619.16} C_VEL
LIN {X 0,Y 144.092,Z 1150.104,A -85,B 0,C 180,E1 2612.386,E2 2612.386} C_VEL
LIN {X 0,Y 144.115,Z 1150.05,A -85,B 0,C 180,E1 2606.42,E2 2606.42} C_VEL
LIN {X 0,Y 144.735,Z 1149.053,A -85,B 0,C 180,E1 2598.807,E2 2598.807} C_VEL
LIN {X 0,Y 146.912,Z 1146.51,A -85,B 0,C 180,E1 2590.519,E2 2590.519} C_VEL
LIN {X 0,Y 151.561,Z 1142.396,A -85,B 0,C 180,E1 2582.07,E2 2582.07} C_VEL
LIN {X 0,Y 158.783,Z 1136.55,A -85,B 0,C 180,E1 2574.153,E2 2574.153} C_VEL
LIN {X 0,Y 168.462,Z 1128.896,A -85,B 0,C 180,E1 2566.957,E2 2566.957} C_VEL
LIN {X 0,Y 179.748,Z 1119.839,A -85,B 0,C 180,E1 2560.842,E2 2560.842} C_VEL
LIN {X 0,Y 192.077,Z 1109.304,A -85,B 0,C 180,E1 2555.702,E2 2555.702} C_VEL
LIN {X 0,Y 202.255,Z 1100.067,A -85,B 0,C 180,E1 2552.195,E2 2552.195} C_VEL
LIN {X 0,Y 186.276,Z 1103.524,A -85,B 0,C 180,E1 2546.114,E2 2546.114} C_VEL
LIN {X 0,Y 174.826,Z 1105.909,A -85,B 0,C 180,E1 2539.374,E2 2539.374} C_VEL
LIN {X 0,Y 169.012,Z 1107.283,A -85,B 0,C 180,E1 2534.388,E2 2534.388} C_VEL
LIN {X 0,Y 164.44,Z 1108.625,A -85,B 0,C 180,E1 2528.392,E2 2528.392} C_VEL
LIN {X 0,Y 161.65,Z 1110.126,A -85,B 0,C 180,E1 2520.71,E2 2520.71} C_VEL
LIN {X 0,Y 163.472,Z 1112.196,A -85,B 0,C 180,E1 2508.714,E2 2508.714} C_VEL
LIN {X 0,Y 171.06,Z 1113.056,A -85,B 0,C 180,E1 2499.828,E2 2499.828} C_VEL
LIN {X 0,Y 179.833,Z 1113.234,A -85,B 0,C 180,E1 2493.946,E2 2493.946} C_VEL
LIN {X 0,Y 192.44,Z 1112.8,A -85,B 0,C 180,E1 2488.255,E2 2488.255} C_VEL
LIN {X 0,Y 180.061,Z 1124.109,A -85,B 0,C 180,E1 2483.094,E2 2483.094} C_VEL
LIN {X 0,Y 170.613,Z 1132.534,A -85,B 0,C 180,E1 2478.109,E2 2478.109} C_VEL
LIN {X 0,Y 166.373,Z 1135.661,A -85,B 0,C 180,E1 2476.169,E2 2476.169} C_VEL
LIN {X 0,Y 152.571,Z 1143.133,A -85,B 0,C 180,E1 2471.007,E2 2471.007} C_VEL
LIN {X 0,Y 149.452,Z 1145.155,A -85,B 0,C 180,E1 2468.907,E2 2468.907} C_VEL
LIN {X 0,Y 142.629,Z 1151.212,A -85,B 0,C 180,E1 2460.78,E2 2460.78} C_VEL
LIN {X 0,Y 138.166,Z 1155.862,A -85,B 0,C 180,E1 2451.658,E2 2451.658} C_VEL
LIN {X 0,Y 136.336,Z 1158.712,A -85,B 0,C 180,E1 2443.141,E2 2443.141} C_VEL
LIN {X 0,Y 136.02,Z 1160.103,A -85,B 0,C 180,E1 2435.484,E2 2435.484} C_VEL
LIN {X 0,Y 136.06,Z 1160.377,A -85,B 0,C 180,E1 2429.158,E2 2429.158} C_VEL
LIN {X 0,Y 136.021,Z 1159.788,A -85,B 0,C 180,E1 2422.397,E2 2422.397} C_VEL
LIN {X 0,Y 136.549,Z 1158.2,A -85,B 0,C 180,E1 2415.134,E2 2415.134} C_VEL
LIN {X 0,Y 138.766,Z 1155.153,A -85,B 0,C 180,E1 2406.653,E2 2406.653} C_VEL
LIN {X 0,Y 143.744,Z 1150.103,A -85,B 0,C 180,E1 2397.615,E2 2397.615} C_VEL
LIN {X 0,Y 151.498,Z 1143.428,A -85,B 0,C 180,E1 2389.203,E2 2389.203} C_VEL
LIN {X 0,Y 161.337,Z 1135.236,A -85,B 0,C 180,E1 2381.954,E2 2381.954} C_VEL
LIN {X 0,Y 173.895,Z 1124.774,A -85,B 0,C 180,E1 2375.267,E2 2375.267} C_VEL
LIN {X 0,Y 186.992,Z 1113.436,A -85,B 0,C 180,E1 2369.977,E2 2369.977} C_VEL
LIN {X 0,Y 200.667,Z 1100.614,A -85,B 0,C 180,E1 2365.595,E2 2365.595} C_VEL
LIN {X 0,Y 215.345,Z 1085.752,A -85,B 0,C 180,E1 2361.78,E2 2361.78} C_VEL
LIN {X 0,Y 228.712,Z 1070.852,A -85,B 0,C 180,E1 2358.874,E2 2358.874} C_VEL
LIN {X 0,Y 242.258,Z 1053.994,A -85,B 0,C 180,E1 2356.344,E2 2356.344} C_VEL
LIN {X 0,Y 254.863,Z 1036.535,A -85,B 0,C 180,E1 2354.3,E2 2354.3} C_VEL
LIN {X 0,Y 266.409,Z 1018.215,A -85,B 0,C 180,E1 2352.628,E2 2352.628} C_VEL
LIN {X 0,Y 277.711,Z 997.679,A -85,B 0,C 180,E1 2351.157,E2 2351.157} C_VEL
LIN {X 0,Y 286.923,Z 978.187,A -85,B 0,C 180,E1 2350.061,E2 2350.061} C_VEL
LIN {X 0,Y 295.157,Z 957.245,A -85,B 0,C 180,E1 2349.139,E2 2349.139} C_VEL
LIN {X 0,Y 302.199,Z 935.486,A -85,B 0,C 180,E1 2348.397,E2 2348.397} C_VEL
LIN {X 0,Y 307.644,Z 913.5,A -85,B 0,C 180,E1 2347.847,E2 2347.847} C_VEL
LIN {X 0,Y 311.786,Z 889.765,A -85,B 0,C 180,E1 2347.378,E2 2347.378} C_VEL
LIN {X 0,Y 326.074,Z 762.782,A -85,B 0,C 180,E1 2345.189,E2 2345.189} C_VEL
LIN {X 0,Y 324.982,Z 760.213,A -85,B 0,C 180,E1 2342.998,E2 2342.998} C_VEL
LIN {X 0,Y 323.89,Z 757.765,A -85,B 0,C 180,E1 2338.584,E2 2338.584} C_VEL
LIN {X 0,Y 323.911,Z 759.313,A -85,B 0,C 180,E1 2335.219,E2 2335.219} C_VEL
LIN {X 0,Y 324.437,Z 760.953,A -85,B 0,C 180,E1 2333.096,E2 2333.096} C_VEL
LIN {X 0,Y 325.516,Z 764.394,A -85,B 0,C 180,E1 2330.503,E2 2330.503} C_VEL
LIN {X 0,Y 310.97,Z 894.967,A -85,B 0,C 180,E1 2328.339,E2 2328.339} C_VEL
LIN {X 0,Y 306.716,Z 917.548,A -85,B 0,C 180,E1 2327.895,E2 2327.895} C_VEL
LIN {X 0,Y 300.967,Z 939.7,A -85,B 0,C 180,E1 2327.334,E2 2327.334} C_VEL
LIN {X 0,Y 293.953,Z 960.679,A -85,B 0,C 180,E1 2326.609,E2 2326.609} C_VEL
LIN {X 0,Y 285.356,Z 981.587,A -85,B 0,C 180,E1 2325.657,E2 2325.657} C_VEL
LIN {X 0,Y 275.956,Z 1000.983,A -85,B 0,C 180,E1 2324.534,E2 2324.534} C_VEL
LIN {X 0,Y 265.033,Z 1020.03,A -85,B 0,C 180,E1 2323.112,E2 2323.112} C_VEL
LIN {X 0,Y 252.335,Z 1039.288,A -85,B 0,C 180,E1 2321.266,E2 2321.266} C_VEL
LIN {X 0,Y 239.643,Z 1056.26,A -85,B 0,C 180,E1 2319.163,E2 2319.163} C_VEL
LIN {X 0,Y 226.489,Z 1071.677,A -85,B 0,C 180,E1 2316.67,E2 2316.67} C_VEL
LIN {X 0,Y 212.271,Z 1086.693,A -85,B 0,C 180,E1 2313.503,E2 2313.503} C_VEL
LIN {X 0,Y 198.79,Z 1099.583,A -85,B 0,C 180,E1 2309.896,E2 2309.896} C_VEL
LIN {X 0,Y 185.281,Z 1111.268,A -85,B 0,C 180,E1 2305.484,E2 2305.484} C_VEL
LIN {X 0,Y 172.18,Z 1121.841,A -85,B 0,C 180,E1 2300.044,E2 2300.044} C_VEL
LIN {X 0,Y 160.598,Z 1130.62,A -85,B 0,C 180,E1 2293.715,E2 2293.715} C_VEL
LIN {X 0,Y 150.668,Z 1137.902,A -85,B 0,C 180,E1 2286.201,E2 2286.201} C_VEL
LIN {X 0,Y 143.311,Z 1143.492,A -85,B 0,C 180,E1 2277.869,E2 2277.869} C_VEL
LIN {X 0,Y 138.802,Z 1147.208,A -85,B 0,C 180,E1 2269.322,E2 2269.322} C_VEL
LIN {X 0,Y 136.582,Z 1149.587,A -85,B 0,C 180,E1 2260.119,E2 2260.119} C_VEL
LIN {X 0,Y 136.105,Z 1150.374,A -85,B 0,C 180,E1 2252.948,E2 2252.948} C_VEL
LIN {X 0,Y 136.114,Z 1150.362,A -85,B 0,C 180,E1 2246.631,E2 2246.631} C_VEL
LIN {X 0,Y 136.697,Z 1149.487,A -85,B 0,C 180,E1 2239.037,E2 2239.037} C_VEL
LIN {X 0,Y 139.107,Z 1146.956,A -85,B 0,C 180,E1 2229.817,E2 2229.817} C_VEL
LIN {X 0,Y 144.101,Z 1142.937,A -85,B 0,C 180,E1 2220.941,E2 2220.941} C_VEL
LIN {X 0,Y 151.804,Z 1137.138,A -85,B 0,C 180,E1 2212.702,E2 2212.702} C_VEL
LIN {X 0,Y 162.427,Z 1129.299,A -85,B 0,C 180,E1 2205.066,E2 2205.066} C_VEL
LIN {X 0,Y 173.892,Z 1120.644,A -85,B 0,C 180,E1 2199.082,E2 2199.082} C_VEL
LIN {X 0,Y 186.74,Z 1110.169,A -85,B 0,C 180,E1 2193.91,E2 2193.91} C_VEL
LIN {X 0,Y 192.306,Z 1105.351,A -85,B 0,C 180,E1 2191.95,E2 2191.95} C_VEL
LIN {X 0,Y 176.942,Z 1108.465,A -85,B 0,C 180,E1 2185.434,E2 2185.434} C_VEL
LIN {X 0,Y 163.935,Z 1111.119,A -85,B 0,C 180,E1 2176.659,E2 2176.659} C_VEL
LIN {X 0,Y 154.794,Z 1114.052,A -85,B 0,C 180,E1 2161.482,E2 2161.482} C_VEL
LIN {X 0,Y 156.863,Z 1116.233,A -85,B 0,C 180,E1 2147.859,E2 2147.859} C_VEL
LIN {X 0,Y 164.971,Z 1117.062,A -85,B 0,C 180,E1 2138.677,E2 2138.677} C_VEL
LIN {X 0,Y 174.151,Z 1117.231,A -85,B 0,C 180,E1 2132.659,E2 2132.659} C_VEL
LIN {X 0,Y 182.92,Z 1117.078,A -85,B 0,C 180,E1 2128.508,E2 2128.508} C_VEL
LIN {X 0,Y 169.673,Z 1128.431,A -85,B 0,C 180,E1 2122.706,E2 2122.706} C_VEL
LIN {X 0,Y 158.796,Z 1137.41,A -85,B 0,C 180,E1 2116.394,E2 2116.394} C_VEL
LIN {X 0,Y 149.452,Z 1145.155,A -85,B 0,C 180,E1 2108.907,E2 2108.907} C_VEL
LIN {X 0,Y 145.922,Z 1147.467,A -85,B 0,C 180,E1 2106.365,E2 2106.365} C_VEL
LIN {X 0,Y 134.289,Z 1152.62,A -85,B 0,C 180,E1 2099.387,E2 2099.387} C_VEL
LIN {X 0,Y 132.121,Z 1153.987,A -85,B 0,C 180,E1 2096.742,E2 2096.742} C_VEL
LIN {X 0,Y 128.917,Z 1157.557,A -85,B 0,C 180,E1 2087.141,E2 2087.141} C_VEL
LIN {X 0,Y 128.086,Z 1159.283,A -85,B 0,C 180,E1 2079.435,E2 2079.435} C_VEL
LIN {X 0,Y 128.046,Z 1159.992,A -85,B 0,C 180,E1 2072.685,E2 2072.685} C_VEL
LIN {X 0,Y 128.04,Z 1159.964,A -85,B 0,C 180,E1 2066.867,E2 2066.867} C_VEL
LIN {X 0,Y 128.099,Z 1159.198,A -85,B 0,C 180,E1 2060.112,E2 2060.112} C_VEL
LIN {X 0,Y 129.204,Z 1157.169,A -85,B 0,C 180,E1 2051.501,E2 2051.501} C_VEL
LIN {X 0,Y 132.911,Z 1153.18,A -85,B 0,C 180,E1 2041.71,E2 2041.71} C_VEL
LIN {X 0,Y 139.531,Z 1147.62,A -85,B 0,C 180,E1 2032.475,E2 2032.475} C_VEL
LIN {X 0,Y 148.647,Z 1140.449,A -85,B 0,C 180,E1 2024.389,E2 2024.389} C_VEL
LIN {X 0,Y 161.049,Z 1130.893,A -85,B 0,C 180,E1 2016.785,E2 2016.785} C_VEL
LIN {X 0,Y 174.517,Z 1120.197,A -85,B 0,C 180,E1 2010.751,E2 2010.751} C_VEL
LIN {X 0,Y 188.818,Z 1107.912,A -85,B 0,C 180,E1 2005.814,E2 2005.814} C_VEL
LIN {X 0,Y 204.282,Z 1093.519,A -85,B 0,C 180,E1 2001.572,E2 2001.572} C_VEL
LIN {X 0,Y 219.019,Z 1078.468,A -85,B 0,C 180,E1 1998.275,E2 1998.275} C_VEL
LIN {X 0,Y 233.077,Z 1062.314,A -85,B 0,C 180,E1 1995.62,E2 1995.62} C_VEL
LIN {X 0,Y 247.196,Z 1044.146,A -85,B 0,C 180,E1 1993.329,E2 1993.329} C_VEL
LIN {X 0,Y 259.744,Z 1025.897,A -85,B 0,C 180,E1 1991.546,E2 1991.546} C_VEL
LIN {X 0,Y 271.154,Z 1006.64,A -85,B 0,C 180,E1 1990.086,E2 1990.086} C_VEL
LIN {X 0,Y 281.82,Z 985.832,A -85,B 0,C 180,E1 1988.853,E2 1988.853} C_VEL
LIN {X 0,Y 290.72,Z 965.242,A -85,B 0,C 180,E1 1987.901,E2 1987.901} C_VEL
LIN {X 0,Y 298.27,Z 943.804,A -85,B 0,C 180,E1 1987.137,E2 1987.137} C_VEL
LIN {X 0,Y 304.522,Z 921.645,A -85,B 0,C 180,E1 1986.547,E2 1986.547} C_VEL
LIN {X 0,Y 309.079,Z 899.439,A -85,B 0,C 180,E1 1986.094,E2 1986.094} C_VEL
LIN {X 0,Y 313.13,Z 868.444,A -85,B 0,C 180,E1 1985.553,E2 1985.553} C_VEL
LIN {X 0,Y 324.376,Z 769.215,A -85,B 0,C 180,E1 1983.888,E2 1983.888} C_VEL
LIN {X 0,Y 323.768,Z 767.859,A -85,B 0,C 180,E1 1982.477,E2 1982.477} C_VEL
LIN {X 0,Y 322.898,Z 765.707,A -85,B 0,C 180,E1 1978.403,E2 1978.403} C_VEL
LIN {X 0,Y 323.29,Z 768.317,A -85,B 0,C 180,E1 1973.696,E2 1973.696} C_VEL
LIN {X 0,Y 323.91,Z 770.674,A -85,B 0,C 180,E1 1971.809,E2 1971.809} C_VEL
LIN {X 0,Y 309.748,Z 894.97,A -85,B 0,C 180,E1 1969.803,E2 1969.803} C_VEL
LIN {X 0,Y 305.413,Z 917.599,A -85,B 0,C 180,E1 1969.376,E2 1969.376} C_VEL
LIN {X 0,Y 299.48,Z 940.053,A -85,B 0,C 180,E1 1968.834,E2 1968.834} C_VEL
LIN {X 0,Y 292.621,Z 960.283,A -85,B 0,C 180,E1 1968.169,E2 1968.169} C_VEL
LIN {X 0,Y 283.941,Z 981.172,A -85,B 0,C 180,E1 1967.271,E2 1967.271} C_VEL
LIN {X 0,Y 274.382,Z 1000.647,A -85,B 0,C 180,E1 1966.201,E2 1966.201} C_VEL
LIN {X 0,Y 263.58,Z 1019.228,A -85,B 0,C 180,E1 1964.888,E2 1964.888} C_VEL
LIN {X 0,Y 251.181,Z 1037.881,A -85,B 0,C 180,E1 1963.205,E2 1963.205} C_VEL
LIN {X 0,Y 238.953,Z 1054.013,A -85,B 0,C 180,E1 1961.334,E2 1961.334} C_VEL
LIN {X 0,Y 225.062,Z 1070.202,A -85,B 0,C 180,E1 1958.899,E2 1958.899} C_VEL
LIN {X 0,Y 211.162,Z 1084.751,A -85,B 0,C 180,E1 1956.045,E2 1956.045} C_VEL
LIN {X 0,Y 197.089,Z 1097.845,A -85,B 0,C 180,E1 1952.598,E2 1952.598} C_VEL
LIN {X 0,Y 182.398,Z 1110.286,A -85,B 0,C 180,E1 1948.176,E2 1948.176} C_VEL
LIN {X 0,Y 168.936,Z 1120.781,A -85,B 0,C 180,E1 1943.035,E2 1943.035} C_VEL
LIN {X 0,Y 156.408,Z 1129.746,A -85,B 0,C 180,E1 1936.783,E2 1936.783} C_VEL
LIN {X 0,Y 144.853,Z 1137.718,A -85,B 0,C 180,E1 1928.739,E2 1928.739} C_VEL
LIN {X 0,Y 136.755,Z 1143.386,A -85,B 0,C 180,E1 1920.297,E2 1920.297} C_VEL
LIN {X 0,Y 131.357,Z 1147.344,A -85,B 0,C 180,E1 1910.962,E2 1910.962} C_VEL
LIN {X 0,Y 128.732,Z 1149.817,A -85,B 0,C 180,E1 1901.196,E2 1901.196} C_VEL
LIN {X 0,Y 128.125,Z 1150.644,A -85,B 0,C 180,E1 1893.579,E2 1893.579} C_VEL
LIN {X 0,Y 128.106,Z 1150.694,A -85,B 0,C 180,E1 1887.316,E2 1887.316} C_VEL
LIN {X 0,Y 128.53,Z 1150.03,A -85,B 0,C 180,E1 1880.146,E2 1880.146} C_VEL
LIN {X 0,Y 130.654,Z 1148.005,A -85,B 0,C 180,E1 1870.788,E2 1870.788} C_VEL
LIN {X 0,Y 135.411,Z 1144.323,A -85,B 0,C 180,E1 1861.486,E2 1861.486} C_VEL
LIN {X 0,Y 143.646,Z 1138.6,A -85,B 0,C 180,E1 1852.227,E2 1852.227} C_VEL
LIN {X 0,Y 154.161,Z 1131.457,A -85,B 0,C 180,E1 1844.484,E2 1844.484} C_VEL
LIN {X 0,Y 166.318,Z 1122.744,A -85,B 0,C 180,E1 1838.044,E2 1838.044} C_VEL
LIN {X 0,Y 180.197,Z 1112.154,A -85,B 0,C 180,E1 1832.498,E2 1832.498} C_VEL
LIN {X 0,Y 182.426,Z 1110.311,A -85,B 0,C 180,E1 1831.655,E2 1831.655} C_VEL
LIN {X 0,Y 165.378,Z 1113.506,A -85,B 0,C 180,E1 1823.518,E2 1823.518} C_VEL
LIN {X 0,Y 151.751,Z 1116.429,A -85,B 0,C 180,E1 1811.017,E2 1811.017} C_VEL
LIN {X 0,Y 149.083,Z 1119.866,A -85,B 0,C 180,E1 1789.177,E2 1789.177} C_VEL
LIN {X 0,Y 157.225,Z 1120.883,A -85,B 0,C 180,E1 1778.748,E2 1778.748} C_VEL
LIN {X 0,Y 167.95,Z 1121.143,A -85,B 0,C 180,E1 1771.56,E2 1771.56} C_VEL
LIN {X 0,Y 173.488,Z 1121.091,A -85,B 0,C 180,E1 1768.853,E2 1768.853} C_VEL
LIN {X 0,Y 160.462,Z 1131.448,A -85,B 0,C 180,E1 1762.9,E2 1762.9} C_VEL
LIN {X 0,Y 148.535,Z 1140.601,A -85,B 0,C 180,E1 1755.524,E2 1755.524} C_VEL
LIN {X 0,Y 139.156,Z 1147.972,A -85,B 0,C 180,E1 1747.105,E2 1747.105} C_VEL
LIN {X 0,Y 132.682,Z 1153.431,A -85,B 0,C 180,E1 1737.854,E2 1737.854} C_VEL
LIN {X 0,Y 132.121,Z 1153.987,A -85,B 0,C 180,E1 1736.742,E2 1736.742} C_VEL
LIN {X 0,Y 129.757,Z 1155.464,A -85,B 0,C 180,E1 1733.572,E2 1733.572} C_VEL
LIN {X 0,Y 123.567,Z 1157.505,A -85,B 0,C 180,E1 1727.671,E2 1727.671} C_VEL
LIN {X 0,Y 120.437,Z 1158.555,A -85,B 0,C 180,E1 1722.907,E2 1722.907} C_VEL
LIN {X 0,Y 120.182,Z 1158.754,A -85,B 0,C 180,E1 1721.583,E2 1721.583} C_VEL
LIN {X 0,Y 120.038,Z 1159.625,A -85,B 0,C 180,E1 1714.299,E2 1714.299} C_VEL
LIN {X 0,Y 120.062,Z 1159.737,A -85,B 0,C 180,E1 1707.882,E2 1707.882} C_VEL
LIN {X 0,Y 120.079,Z 1159.127,A -85,B 0,C 180,E1 1700.897,E2 1700.897} C_VEL
LIN {X 0,Y 120.919,Z 1157.488,A -85,B 0,C 180,E1 1692.682,E2 1692.682} C_VEL
LIN {X 0,Y 124.212,Z 1154.19,A -85,B 0,C 180,E1 1682.688,E2 1682.688} C_VEL
LIN {X 0,Y 130.698,Z 1148.956,A -85,B 0,C 180,E1 1672.817,E2 1672.817} C_VEL
LIN {X 0,Y 140.726,Z 1141.702,A -85,B 0,C 180,E1 1663.555,E2 1663.555} C_VEL
LIN {X 0,Y 152.582,Z 1133.254,A -85,B 0,C 180,E1 1656.139,E2 1656.139} C_VEL
LIN {X 0,Y 166.137,Z 1123.08,A -85,B 0,C 180,E1 1649.93,E2 1649.93} C_VEL
LIN {X 0,Y 180.711,Z 1111.5,A -85,B 0,C 180,E1 1644.851,E2 1644.851} C_VEL
LIN {X 0,Y 194.831,Z 1099.235,A -85,B 0,C 180,E1 1640.93,E2 1640.93} C_VEL
LIN {X 0,Y 210.565,Z 1084.193,A -85,B 0,C 180,E1 1637.361,E2 1637.361} C_VEL
LIN {X 0,Y 225.244,Z 1068.651,A -85,B 0,C 180,E1 1634.601,E2 1634.601} C_VEL
LIN {X 0,Y 239.472,Z 1051.528,A -85,B 0,C 180,E1 1632.309,E2 1632.309} C_VEL
LIN {X 0,Y 253.124,Z 1032.959,A -85,B 0,C 180,E1 1630.4,E2 1630.4} C_VEL
LIN {X 0,Y 265.36,Z 1013.996,A -85,B 0,C 180,E1 1628.886,E2 1628.886} C_VEL
LIN {X 0,Y 276.421,Z 993.864,A -85,B 0,C 180,E1 1627.648,E2 1627.648} C_VEL
LIN {X 0,Y 286.528,Z 972.217,A -85,B 0,C 180,E1 1626.612,E2 1626.612} C_VEL
LIN {X 0,Y 294.631,Z 951.355,A -85,B 0,C 180,E1 1625.843,E2 1625.843} C_VEL
LIN {X 0,Y 301.249,Z 929.837,A -85,B 0,C 180,E1 1625.241,E2 1625.241} C_VEL
LIN {X 0,Y 306.64,Z 907.067,A -85,B 0,C 180,E1 1624.758,E2 1624.758} C_VEL
LIN {X 0,Y 310.231,Z 884.664,A -85,B 0,C 180,E1 1624.361,E2 1624.361} C_VEL
LIN {X 0,Y 322.814,Z 775.901,A -85,B 0,C 180,E1 1622.574,E2 1622.574} C_VEL
LIN {X 0,Y 321.918,Z 773.651,A -85,B 0,C 180,E1 1618.398,E2 1618.398} C_VEL
LIN {X 0,Y 322.264,Z 776.244,A -85,B 0,C 180,E1 1613.855,E2 1613.855} C_VEL
LIN {X 0,Y 322.432,Z 777.302,A -85,B 0,C 180,E1 1613.123,E2 1613.123} C_VEL
LIN {X 0,Y 308.732,Z 894.945,A -85,B 0,C 180,E1 1611.277,E2 1611.277} C_VEL
LIN {X 0,Y 304.345,Z 917.517,A -85,B 0,C 180,E1 1610.871,E2 1610.871} C_VEL
LIN {X 0,Y 298.607,Z 939.141,A -85,B 0,C 180,E1 1610.382,E2 1610.382} C_VEL
LIN {X 0,Y 291.613,Z 959.599,A -85,B 0,C 180,E1 1609.752,E2 1609.752} C_VEL
LIN {X 0,Y 282.753,Z 980.757,A -85,B 0,C 180,E1 1608.898,E2 1608.898} C_VEL
LIN {X 0,Y 273.043,Z 1000.291,A -85,B 0,C 180,E1 1607.886,E2 1607.886} C_VEL
LIN {X 0,Y 262.055,Z 1018.95,A -85,B 0,C 180,E1 1606.642,E2 1606.642} C_VEL
LIN {X 0,Y 249.87,Z 1037.074,A -85,B 0,C 180,E1 1605.099,E2 1605.099} C_VEL
LIN {X 0,Y 237.731,Z 1052.839,A -85,B 0,C 180,E1 1603.381,E2 1603.381} C_VEL
LIN {X 0,Y 223.128,Z 1069.636,A -85,B 0,C 180,E1 1601,E2 1601} C_VEL
LIN {X 0,Y 208.82,Z 1084.296,A -85,B 0,C 180,E1 1598.264,E2 1598.264} C_VEL
LIN {X 0,Y 194.256,Z 1097.477,A -85,B 0,C 180,E1 1594.944,E2 1594.944} C_VEL
LIN {X 0,Y 178.958,Z 1110.034,A -85,B 0,C 180,E1 1590.644,E2 1590.644} C_VEL
LIN {X 0,Y 164.812,Z 1120.587,A -85,B 0,C 180,E1 1585.595,E2 1585.595} C_VEL
LIN {X 0,Y 151.499,Z 1129.658,A -85,B 0,C 180,E1 1579.374,E2 1579.374} C_VEL
LIN {X 0,Y 139.673,Z 1137.334,A -85,B 0,C 180,E1 1571.74,E2 1571.74} C_VEL
LIN {X 0,Y 130.458,Z 1143.201,A -85,B 0,C 180,E1 1562.967,E2 1562.967} C_VEL
LIN {X 0,Y 124.216,Z 1147.338,A -85,B 0,C 180,E1 1553.23,E2 1553.23} C_VEL
LIN {X 0,Y 121.071,Z 1149.907,A -85,B 0,C 180,E1 1543.37,E2 1543.37} C_VEL
LIN {X 0,Y 120.15,Z 1150.915,A -85,B 0,C 180,E1 1534.295,E2 1534.295} C_VEL
LIN {X 0,Y 120.111,Z 1150.995,A -85,B 0,C 180,E1 1527.376,E2 1527.376} C_VEL
LIN {X 0,Y 120.608,Z 1150.322,A -85,B 0,C 180,E1 1519.491,E2 1519.491} C_VEL
LIN {X 0,Y 123.016,Z 1148.301,A -85,B 0,C 180,E1 1509.543,E2 1509.543} C_VEL
LIN {X 0,Y 128.402,Z 1144.551,A -85,B 0,C 180,E1 1499.592,E2 1499.592} C_VEL
LIN {X 0,Y 137.262,Z 1138.899,A -85,B 0,C 180,E1 1490.132,E2 1490.132} C_VEL
LIN {X 0,Y 148.529,Z 1131.758,A -85,B 0,C 180,E1 1482.226,E2 1482.226} C_VEL
LIN {X 0,Y 161.395,Z 1123.045,A -85,B 0,C 180,E1 1475.751,E2 1475.751} C_VEL
LIN {X 0,Y 172.555,Z 1115.032,A -85,B 0,C 180,E1 1471.337,E2 1471.337} C_VEL
LIN {X 0,Y 157.037,Z 1117.652,A -85,B 0,C 180,E1 1463.252,E2 1463.252} C_VEL
LIN {X 0,Y 145.015,Z 1120.064,A -85,B 0,C 180,E1 1451.939,E2 1451.939} C_VEL
LIN {X 0,Y 142.102,Z 1123.539,A -85,B 0,C 180,E1 1428.639,E2 1428.639} C_VEL
LIN {X 0,Y 150.623,Z 1124.561,A -85,B 0,C 180,E1 1417.768,E2 1417.768} C_VEL
LIN {X 0,Y 161.717,Z 1124.838,A -85,B 0,C 180,E1 1410.356,E2 1410.356} C_VEL
LIN {X 0,Y 164.019,Z 1124.814,A -85,B 0,C 180,E1 1409.2,E2 1409.2} C_VEL
LIN {X 0,Y 150.04,Z 1135.109,A -85,B 0,C 180,E1 1402.468,E2 1402.468} C_VEL
LIN {X 0,Y 138.766,Z 1143.232,A -85,B 0,C 180,E1 1394.921,E2 1394.921} C_VEL
LIN {X 0,Y 129.629,Z 1149.804,A -85,B 0,C 180,E1 1385.888,E2 1385.888} C_VEL
LIN {X 0,Y 123.364,Z 1154.921,A -85,B 0,C 180,E1 1375.44,E2 1375.44} C_VEL
LIN {X 0,Y 120.744,Z 1157.752,A -85,B 0,C 180,E1 1366.353,E2 1366.353} C_VEL
LIN {X 0,Y 120.182,Z 1158.754,A -85,B 0,C 180,E1 1361.583,E2 1361.583} C_VEL
LIN {X 0,Y 119.145,Z 1159.277,A -85,B 0,C 180,E1 1358.176,E2 1358.176} C_VEL
LIN {X 0,Y 116.174,Z 1159.535,A -85,B 0,C 180,E1 1353.494,E2 1353.494} C_VEL
LIN {X 0,Y 112.232,Z 1159.379,A -85,B 0,C 180,E1 1346.027,E2 1346.027} C_VEL
LIN {X 0,Y 112.032,Z 1159.273,A -85,B 0,C 180,E1 1344.286,E2 1344.286} C_VEL
LIN {X 0,Y 112.513,Z 1158.049,A -85,B 0,C 180,E1 1335.066,E2 1335.066} C_VEL
LIN {X 0,Y 115.113,Z 1155.278,A -85,B 0,C 180,E1 1324.811,E2 1324.811} C_VEL
LIN {X 0,Y 120.789,Z 1151.04,A -85,B 0,C 180,E1 1314.589,E2 1314.589} C_VEL
LIN {X 0,Y 129.936,Z 1144.783,A -85,B 0,C 180,E1 1304.932,E2 1304.932} C_VEL
LIN {X 0,Y 141.984,Z 1136.829,A -85,B 0,C 180,E1 1296.602,E2 1296.602} C_VEL
LIN {X 0,Y 154.998,Z 1127.896,A -85,B 0,C 180,E1 1290.185,E2 1290.185} C_VEL
LIN {X 0,Y 170.336,Z 1116.609,A -85,B 0,C 180,E1 1284.516,E2 1284.516} C_VEL
LIN {X 0,Y 185.517,Z 1104.533,A -85,B 0,C 180,E1 1280.177,E2 1280.177} C_VEL
LIN {X 0,Y 200.454,Z 1091.27,A -85,B 0,C 180,E1 1276.726,E2 1276.726} C_VEL
LIN {X 0,Y 216.151,Z 1075.866,A -85,B 0,C 180,E1 1273.734,E2 1273.734} C_VEL
LIN {X 0,Y 230.077,Z 1060.545,A -85,B 0,C 180,E1 1271.486,E2 1271.486} C_VEL
LIN {X 0,Y 244.314,Z 1042.8,A -85,B 0,C 180,E1 1269.495,E2 1269.495} C_VEL
LIN {X 0,Y 256.935,Z 1025.032,A -85,B 0,C 180,E1 1267.949,E2 1267.949} C_VEL
LIN {X 0,Y 268.291,Z 1006.472,A -85,B 0,C 180,E1 1266.692,E2 1266.692} C_VEL
LIN {X 0,Y 279.29,Z 985.662,A -85,B 0,C 180,E1 1265.589,E2 1265.589} C_VEL
LIN {X 0,Y 287.978,Z 966.169,A -85,B 0,C 180,E1 1264.779,E2 1264.779} C_VEL
LIN {X 0,Y 295.716,Z 945.07,A -85,B 0,C 180,E1 1264.099,E2 1264.099} C_VEL
LIN {X 0,Y 302.17,Z 923.183,A -85,B 0,C 180,E1 1263.572,E2 1263.572} C_VEL
LIN {X 0,Y 307.046,Z 900.256,A -85,B 0,C 180,E1 1263.145,E2 1263.145} C_VEL
LIN {X 0,Y 311.151,Z 870.215,A -85,B 0,C 180,E1 1262.654,E2 1262.654} C_VEL
LIN {X 0,Y 321.367,Z 783.047,A -85,B 0,C 180,E1 1261.247,E2 1261.247} C_VEL
LIN {X 0,Y 320.933,Z 781.596,A -85,B 0,C 180,E1 1258.393,E2 1258.393} C_VEL
LIN {X 0,Y 321.122,Z 783.896,A -85,B 0,C 180,E1 1254.448,E2 1254.448} C_VEL
LIN {X 0,Y 307.913,Z 894.985,A -85,B 0,C 180,E1 1252.76,E2 1252.76} C_VEL
LIN {X 0,Y 303.456,Z 917.564,A -85,B 0,C 180,E1 1252.373,E2 1252.373} C_VEL
LIN {X 0,Y 297.429,Z 939.843,A -85,B 0,C 180,E1 1251.897,E2 1251.897} C_VEL
LIN {X 0,Y 290.301,Z 960.331,A -85,B 0,C 180,E1 1251.3,E2 1251.3} C_VEL
LIN {X 0,Y 281.324,Z 981.335,A -85,B 0,C 180,E1 1250.495,E2 1250.495} C_VEL
LIN {X 0,Y 271.476,Z 1000.808,A -85,B 0,C 180,E1 1249.539,E2 1249.539} C_VEL
LIN {X 0,Y 260.316,Z 1019.399,A -85,B 0,C 180,E1 1248.363,E2 1248.363} C_VEL
LIN {X 0,Y 247.463,Z 1038.071,A -85,B 0,C 180,E1 1246.843,E2 1246.843} C_VEL
LIN {X 0,Y 234.802,Z 1054.128,A -85,B 0,C 180,E1 1245.159,E2 1245.159} C_VEL
LIN {X 0,Y 220.621,Z 1069.984,A -85,B 0,C 180,E1 1242.992,E2 1242.992} C_VEL
LIN {X 0,Y 205.948,Z 1084.63,A -85,B 0,C 180,E1 1240.366,E2 1240.366} C_VEL
LIN {X 0,Y 190.945,Z 1097.798,A -85,B 0,C 180,E1 1237.162,E2 1237.162} C_VEL
LIN {X 0,Y 175.095,Z 1110.342,A -85,B 0,C 180,E1 1232.977,E2 1232.977} C_VEL
LIN {X 0,Y 160.327,Z 1120.896,A -85,B 0,C 180,E1 1228.011,E2 1228.011} C_VEL
LIN {X 0,Y 146.293,Z 1129.958,A -85,B 0,C 180,E1 1221.812,E2 1221.812} C_VEL
LIN {X 0,Y 133.67,Z 1137.633,A -85,B 0,C 180,E1 1214.079,E2 1214.079} C_VEL
LIN {X 0,Y 123.679,Z 1143.5,A -85,B 0,C 180,E1 1205.029,E2 1205.029} C_VEL
LIN {X 0,Y 116.78,Z 1147.633,A -85,B 0,C 180,E1 1194.805,E2 1194.805} C_VEL
LIN {X 0,Y 113.226,Z 1150.201,A -85,B 0,C 180,E1 1184.315,E2 1184.315} C_VEL
LIN {X 0,Y 112.165,Z 1151.206,A -85,B 0,C 180,E1 1174.602,E2 1174.602} C_VEL
LIN {X 0,Y 112.118,Z 1151.287,A -85,B 0,C 180,E1 1167.22,E2 1167.22} C_VEL
LIN {X 0,Y 112.704,Z 1150.615,A -85,B 0,C 180,E1 1158.745,E2 1158.745} C_VEL
LIN {X 0,Y 115.599,Z 1148.477,A -85,B 0,C 180,E1 1147.745,E2 1147.745} C_VEL
LIN {X 0,Y 121.423,Z 1144.846,A -85,B 0,C 180,E1 1137.639,E2 1137.639} C_VEL
LIN {X 0,Y 131.078,Z 1139.195,A -85,B 0,C 180,E1 1127.835,E2 1127.835} C_VEL
LIN {X 0,Y 143.146,Z 1132.059,A -85,B 0,C 180,E1 1119.795,E2 1119.795} C_VEL
LIN {X 0,Y 157.035,Z 1123.161,A -85,B 0,C 180,E1 1113.202,E2 1113.202} C_VEL
LIN {X 0,Y 162.586,Z 1119.376,A -85,B 0,C 180,E1 1111.011,E2 1111.011} C_VEL
LIN {X 0,Y 144.928,Z 1122.33,A -85,B 0,C 180,E1 1100.18,E2 1100.18} C_VEL
LIN {X 0,Y 133.595,Z 1125.162,A -85,B 0,C 180,E1 1082.146,E2 1082.146} C_VEL
LIN {X 0,Y 135.853,Z 1127.189,A -85,B 0,C 180,E1 1066.379,E2 1066.379} C_VEL
LIN {X 0,Y 145.304,Z 1128.073,A -85,B 0,C 180,E1 1055.616,E2 1055.616} C_VEL
LIN {X 0,Y 154.311,Z 1128.454,A -85,B 0,C 180,E1 1049.517,E2 1049.517} C_VEL
LIN {X 0,Y 140.792,Z 1137.745,A -85,B 0,C 180,E1 1042.692,E2 1042.692} C_VEL
LIN {X 0,Y 128.982,Z 1145.473,A -85,B 0,C 180,E1 1034.241,E2 1034.241} C_VEL
LIN {X 0,Y 119.787,Z 1151.734,A -85,B 0,C 180,E1 1024.004,E2 1024.004} C_VEL
LIN {X 0,Y 114.74,Z 1155.648,A -85,B 0,C 180,E1 1014.178,E2 1014.178} C_VEL
LIN {X 0,Y 112.337,Z 1158.318,A -85,B 0,C 180,E1 1003.381,E2 1003.381} C_VEL
LIN {X 0,Y 112.035,Z 1159.307,A -85,B 0,C 180,E1 995.12,E2 995.12} C_VEL
LIN {X 0,Y 112.073,Z 1159.481,A -85,B 0,C 180,E1 988.466,E2 988.466} C_VEL
LIN {X 0,Y 112.032,Z 1159.273,A -85,B 0,C 180,E1 984.286,E2 984.286} C_VEL
LIN {X 0,Y 111.22,Z 1158.974,A -85,B 0,C 180,E1 980.619,E2 980.619} C_VEL
LIN {X 0,Y 108.372,Z 1158.134,A -85,B 0,C 180,E1 974.985,E2 974.985} C_VEL
LIN {X 0,Y 106.241,Z 1156.659,A -85,B 0,C 180,E1 968.487,E2 968.487} C_VEL
LIN {X 0,Y 106.619,Z 1155.881,A -85,B 0,C 180,E1 965.802,E2 965.802} C_VEL
LIN {X 0,Y 111.931,Z 1152.052,A -85,B 0,C 180,E1 955.131,E2 955.131} C_VEL
LIN {X 0,Y 121.107,Z 1146.381,A -85,B 0,C 180,E1 944.764,E2 944.764} C_VEL
LIN {X 0,Y 132.734,Z 1139.248,A -85,B 0,C 180,E1 936.292,E2 936.292} C_VEL
LIN {X 0,Y 147.337,Z 1129.954,A -85,B 0,C 180,E1 928.905,E2 928.905} C_VEL
LIN {X 0,Y 162.297,Z 1119.795,A -85,B 0,C 180,E1 923.373,E2 923.373} C_VEL
LIN {X 0,Y 178.461,Z 1107.594,A -85,B 0,C 180,E1 918.763,E2 918.763} C_VEL
LIN {X 0,Y 195.577,Z 1093.296,A -85,B 0,C 180,E1 914.93,E2 914.93} C_VEL
LIN {X 0,Y 211.796,Z 1078.137,A -85,B 0,C 180,E1 911.988,E2 911.988} C_VEL
LIN {X 0,Y 226.714,Z 1062.239,A -85,B 0,C 180,E1 909.706,E2 909.706} C_VEL
LIN {X 0,Y 241.902,Z 1043.945,A -85,B 0,C 180,E1 907.718,E2 907.718} C_VEL
LIN {X 0,Y 254.969,Z 1026.001,A -85,B 0,C 180,E1 906.227,E2 906.227} C_VEL
LIN {X 0,Y 266.494,Z 1007.623,A -85,B 0,C 180,E1 905.039,E2 905.039} C_VEL
LIN {X 0,Y 277.122,Z 988.187,A -85,B 0,C 180,E1 904.049,E2 904.049} C_VEL
LIN {X 0,Y 286.419,Z 967.834,A -85,B 0,C 180,E1 903.24,E2 903.24} C_VEL
LIN {X 0,Y 294.755,Z 945.703,A -85,B 0,C 180,E1 902.562,E2 902.562} C_VEL
LIN {X 0,Y 301.367,Z 923.642,A -85,B 0,C 180,E1 902.062,E2 902.062} C_VEL
LIN {X 0,Y 306.305,Z 900.821,A -85,B 0,C 180,E1 901.661,E2 901.661} C_VEL
LIN {X 0,Y 310.493,Z 870.91,A -85,B 0,C 180,E1 901.19,E2 901.19} C_VEL
LIN {X 0,Y 320.1,Z 790.235,A -85,B 0,C 180,E1 899.959,E2 899.959} C_VEL
LIN {X 0,Y 319.937,Z 789.587,A -85,B 0,C 180,E1 898.209,E2 898.209} C_VEL
LIN {X 0,Y 319.906,Z 791.152,A -85,B 0,C 180,E1 895.773,E2 895.773} C_VEL
LIN {X 0,Y 307.302,Z 895.025,A -85,B 0,C 180,E1 894.249,E2 894.249} C_VEL
LIN {X 0,Y 302.776,Z 917.61,A -85,B 0,C 180,E1 893.883,E2 893.883} C_VEL
LIN {X 0,Y 296.592,Z 940.145,A -85,B 0,C 180,E1 893.433,E2 893.433} C_VEL
LIN {X 0,Y 289.683,Z 959.789,A -85,B 0,C 180,E1 892.898,E2 892.898} C_VEL
LIN {X 0,Y 280.593,Z 980.918,A -85,B 0,C 180,E1 892.147,E2 892.147} C_VEL
LIN {X 0,Y 270.61,Z 1000.451,A -85,B 0,C 180,E1 891.254,E2 891.254} C_VEL
LIN {X 0,Y 259.284,Z 1019.12,A -85,B 0,C 180,E1 890.154,E2 890.154} C_VEL
LIN {X 0,Y 246.218,Z 1037.865,A -85,B 0,C 180,E1 888.726,E2 888.726} C_VEL
LIN {X 0,Y 233.064,Z 1054.263,A -85,B 0,C 180,E1 887.109,E2 887.109} C_VEL
LIN {X 0,Y 218.387,Z 1070.332,A -85,B 0,C 180,E1 885.026,E2 885.026} C_VEL
LIN {X 0,Y 203.361,Z 1084.963,A -85,B 0,C 180,E1 882.523,E2 882.523} C_VEL
LIN {X 0,Y 187.819,Z 1098.211,A -85,B 0,C 180,E1 879.429,E2 879.429} C_VEL
LIN {X 0,Y 170.738,Z 1111.21,A -85,B 0,C 180,E1 875.189,E2 875.189} C_VEL
LIN {X 0,Y 155.406,Z 1121.703,A -85,B 0,C 180,E1 870.293,E2 870.293} C_VEL
LIN {X 0,Y 140.711,Z 1130.651,A -85,B 0,C 180,E1 864.102,E2 864.102} C_VEL
LIN {X 0,Y 126.806,Z 1138.515,A -85,B 0,C 180,E1 855.851,E2 855.851} C_VEL
LIN {X 0,Y 116.246,Z 1144.28,A -85,B 0,C 180,E1 846.405,E2 846.405} C_VEL
LIN {X 0,Y 108.924,Z 1148.232,A -85,B 0,C 180,E1 835.558,E2 835.558} C_VEL
LIN {X 0,Y 105.094,Z 1150.696,A -85,B 0,C 180,E1 823.76,E2 823.76} C_VEL
LIN {X 0,Y 104.161,Z 1151.517,A -85,B 0,C 180,E1 814.404,E2 814.404} C_VEL
LIN {X 0,Y 104.131,Z 1151.566,A -85,B 0,C 180,E1 806.697,E2 806.697} C_VEL
LIN {X 0,Y 104.819,Z 1150.907,A -85,B 0,C 180,E1 797.886,E2 797.886} C_VEL
LIN {X 0,Y 108.168,Z 1148.74,A -85,B 0,C 180,E1 786.001,E2 786.001} C_VEL
LIN {X 0,Y 114.603,Z 1145.142,A -85,B 0,C 180,E1 775.452,E2 775.452} C_VEL
LIN {X 0,Y 125.125,Z 1139.494,A -85,B 0,C 180,E1 765.315,E2 765.315} C_VEL
LIN {X 0,Y 138.041,Z 1132.36,A -85,B 0,C 180,E1 757.178,E2 757.178} C_VEL
LIN {X 0,Y 152.735,Z 1123.43,A -85,B 0,C 180,E1 750.597,E2 750.597} C_VEL
LIN {X 0,Y 137.696,Z 1125.755,A -85,B 0,C 180,E1 740.844,E2 740.844} C_VEL
LIN {X 0,Y 126.387,Z 1128.456,A -85,B 0,C 180,E1 722.722,E2 722.722} C_VEL
LIN {X 0,Y 128.799,Z 1130.537,A -85,B 0,C 180,E1 705.618,E2 705.618} C_VEL
LIN {X 0,Y 138.717,Z 1131.428,A -85,B 0,C 180,E1 694.377,E2 694.377} C_VEL
LIN {X 0,Y 144.8,Z 1131.755,A -85,B 0,C 180,E1 689.973,E2 689.973} C_VEL
LIN {X 0,Y 130.923,Z 1140.42,A -85,B 0,C 180,E1 682.585,E2 682.585} C_VEL
LIN {X 0,Y 119.19,Z 1147.591,A -85,B 0,C 180,E1 673.463,E2 673.463} C_VEL
LIN {X 0,Y 110.95,Z 1152.746,A -85,B 0,C 180,E1 663.348,E2 663.348} C_VEL
LIN {X 0,Y 105.668,Z 1156.666,A -85,B 0,C 180,E1 651.074,E2 651.074} C_VEL
LIN {X 0,Y 104.148,Z 1158.476,A -85,B 0,C 180,E1 641.07,E2 641.07} C_VEL
LIN {X 0,Y 104.058,Z 1159.144,A -85,B 0,C 180,E1 632.754,E2 632.754} C_VEL
LIN {X 0,Y 104.048,Z 1159.09,A -85,B 0,C 180,E1 626.143,E2 626.143} C_VEL
LIN {X 0,Y 104.221,Z 1158.313,A -85,B 0,C 180,E1 617.816,E2 617.816} C_VEL
LIN {X 0,Y 106.31,Z 1156.151,A -85,B 0,C 180,E1 606.733,E2 606.733} C_VEL
LIN {X 0,Y 106.619,Z 1155.881,A -85,B 0,C 180,E1 605.802,E2 605.802} C_VEL
LIN {X 0,Y 107.235,Z 1154.633,A -85,B 0,C 180,E1 601.712,E2 601.712} C_VEL
LIN {X 0,Y 107.813,Z 1150.606,A -85,B 0,C 180,E1 589.952,E2 589.952} C_VEL
LIN {X 0,Y 109.579,Z 1149.277,A -85,B 0,C 180,E1 587.251,E2 587.251} C_VEL
LIN {X 0,Y 121.042,Z 1142.903,A -85,B 0,C 180,E1 577.533,E2 577.533} C_VEL
LIN {X 0,Y 134.744,Z 1134.947,A -85,B 0,C 180,E1 569.75,E2 569.75} C_VEL
LIN {X 0,Y 150.363,Z 1125.314,A -85,B 0,C 180,E1 563.415,E2 563.415} C_VEL
LIN {X 0,Y 166.589,Z 1114.206,A -85,B 0,C 180,E1 558.502,E2 558.502} C_VEL
LIN {X 0,Y 183.797,Z 1101.119,A -85,B 0,C 180,E1 554.459,E2 554.459} C_VEL
LIN {X 0,Y 199.93,Z 1087.446,A -85,B 0,C 180,E1 551.418,E2 551.418} C_VEL
LIN {X 0,Y 216.072,Z 1071.848,A -85,B 0,C 180,E1 548.897,E2 548.897} C_VEL
LIN {X 0,Y 232.061,Z 1054.361,A -85,B 0,C 180,E1 546.795,E2 546.795} C_VEL
LIN {X 0,Y 245.986,Z 1037.046,A -85,B 0,C 180,E1 545.219,E2 545.219} C_VEL
LIN {X 0,Y 259.065,Z 1018.156,A -85,B 0,C 180,E1 543.902,E2 543.902} C_VEL
LIN {X 0,Y 271.288,Z 997.72,A -85,B 0,C 180,E1 542.805,E2 542.805} C_VEL
LIN {X 0,Y 281.709,Z 977.188,A -85,B 0,C 180,E1 541.954,E2 541.954} C_VEL
LIN {X 0,Y 290.532,Z 955.973,A -85,B 0,C 180,E1 541.278,E2 541.278} C_VEL
LIN {X 0,Y 298.061,Z 933.639,A -85,B 0,C 180,E1 540.734,E2 540.734} C_VEL
LIN {X 0,Y 303.642,Z 912.057,A -85,B 0,C 180,E1 540.34,E2 540.34} C_VEL
LIN {X 0,Y 307.806,Z 888.944,A -85,B 0,C 180,E1 539.979,E2 539.979} C_VEL
LIN {X 0,Y 318.988,Z 797.511,A -85,B 0,C 180,E1 538.608,E2 538.608} C_VEL
LIN {X 0,Y 318.883,Z 798.24,A -85,B 0,C 180,E1 537.111,E2 537.111} C_VEL
LIN {X 0,Y 306.899,Z 895.065,A -85,B 0,C 180,E1 535.743,E2 535.743} C_VEL
LIN {X 0,Y 302.308,Z 917.666,A -85,B 0,C 180,E1 535.399,E2 535.399} C_VEL
LIN {X 0,Y 296.094,Z 940.071,A -85,B 0,C 180,E1 534.984,E2 534.984} C_VEL
LIN {X 0,Y 288.807,Z 960.52,A -85,B 0,C 180,E1 534.466,E2 534.466} C_VEL
LIN {X 0,Y 279.614,Z 981.497,A -85,B 0,C 180,E1 533.769,E2 533.769} C_VEL
LIN {X 0,Y 269.508,Z 1000.967,A -85,B 0,C 180,E1 532.937,E2 532.937} C_VEL
LIN {X 0,Y 258.032,Z 1019.567,A -85,B 0,C 180,E1 531.912,E2 531.912} C_VEL
LIN {X 0,Y 245.05,Z 1037.901,A -85,B 0,C 180,E1 530.606,E2 530.606} C_VEL
LIN {X 0,Y 231.654,Z 1054.334,A -85,B 0,C 180,E1 529.092,E2 529.092} C_VEL
LIN {X 0,Y 216.434,Z 1070.679,A -85,B 0,C 180,E1 527.099,E2 527.099} C_VEL
LIN {X 0,Y 200.898,Z 1085.44,A -85,B 0,C 180,E1 524.705,E2 524.705} C_VEL
LIN {X 0,Y 184.624,Z 1098.922,A -85,B 0,C 180,E1 521.692,E2 521.692} C_VEL
LIN {X 0,Y 167.472,Z 1111.522,A -85,B 0,C 180,E1 517.729,E2 517.729} C_VEL
LIN {X 0,Y 151.515,Z 1122.009,A -85,B 0,C 180,E1 512.984,E2 512.984} C_VEL
LIN {X 0,Y 136.065,Z 1130.955,A -85,B 0,C 180,E1 506.9,E2 506.9} C_VEL
LIN {X 0,Y 121.242,Z 1138.813,A -85,B 0,C 180,E1 498.631,E2 498.631} C_VEL
LIN {X 0,Y 109.772,Z 1144.578,A -85,B 0,C 180,E1 488.939,E2 488.939} C_VEL
LIN {X 0,Y 101.64,Z 1148.527,A -85,B 0,C 180,E1 477.539,E2 477.539} C_VEL
LIN {X 0,Y 97.265,Z 1150.99,A -85,B 0,C 180,E1 464.892,E2 464.892} C_VEL
LIN {X 0,Y 96.178,Z 1151.809,A -85,B 0,C 180,E1 454.771,E2 454.771} C_VEL
LIN {X 0,Y 96.134,Z 1151.872,A -85,B 0,C 180,E1 446.854,E2 446.854} C_VEL
LIN {X 0,Y 96.858,Z 1151.262,A -85,B 0,C 180,E1 437.48,E2 437.48} C_VEL
LIN {X 0,Y 100.395,Z 1149.272,A -85,B 0,C 180,E1 425.001,E2 425.001} C_VEL
LIN {X 0,Y 107.551,Z 1145.635,A -85,B 0,C 180,E1 413.488,E2 413.488} C_VEL
LIN {X 0,Y 119.437,Z 1139.792,A -85,B 0,C 180,E1 402.55,E2 402.55} C_VEL
LIN {X 0,Y 133.246,Z 1132.661,A -85,B 0,C 180,E1 394.368,E2 394.368} C_VEL
LIN {X 0,Y 142.573,Z 1127.377,A -85,B 0,C 180,E1 390.119,E2 390.119} C_VEL
LIN {X 0,Y 124.673,Z 1130.067,A -85,B 0,C 180,E1 375.348,E2 375.348} C_VEL
LIN {X 0,Y 120.519,Z 1133.377,A -85,B 0,C 180,E1 347.057,E2 347.057} C_VEL
LIN {X 0,Y 130.634,Z 1134.433,A -85,B 0,C 180,E1 334.135,E2 334.135} C_VEL
LIN {X 0,Y 135.365,Z 1134.658,A -85,B 0,C 180,E1 330.539,E2 330.539} C_VEL
LIN {X 0,Y 121.046,Z 1142.963,A -85,B 0,C 180,E1 322.465,E2 322.465} C_VEL
LIN {X 0,Y 109.859,Z 1149.161,A -85,B 0,C 180,E1 313.047,E2 313.047} C_VEL
LIN {X 0,Y 101.106,Z 1154.272,A -85,B 0,C 180,E1 300.646,E2 300.646} C_VEL
LIN {X 0,Y 97.166,Z 1157.107,A -85,B 0,C 180,E1 289.226,E2 289.226} C_VEL
LIN {X 0,Y 96.04,Z 1158.641,A -85,B 0,C 180,E1 277.779,E2 277.779} C_VEL
LIN {X 0,Y 96.087,Z 1158.947,A -85,B 0,C 180,E1 269.404,E2 269.404} C_VEL
LIN {X 0,Y 96.078,Z 1158.542,A -85,B 0,C 180,E1 261.019,E2 261.019} C_VEL
LIN {X 0,Y 97.427,Z 1156.839,A -85,B 0,C 180,E1 249.578,E2 249.578} C_VEL
LIN {X 0,Y 101.82,Z 1153.822,A -85,B 0,C 180,E1 237.976,E2 237.976} C_VEL
LIN {X 0,Y 109.579,Z 1149.277,A -85,B 0,C 180,E1 227.251,E2 227.251} C_VEL
LIN {X 0,Y 112.149,Z 1147.418,A -85,B 0,C 180,E1 223.593,E2 223.593} C_VEL
LIN {X 0,Y 118.114,Z 1141.788,A -85,B 0,C 180,E1 213.516,E2 213.516} C_VEL
LIN {X 0,Y 121.303,Z 1139.817,A -85,B 0,C 180,E1 211.195,E2 211.195} C_VEL
LIN {X 0,Y 136.861,Z 1131.223,A -85,B 0,C 180,E1 204.047,E2 204.047} C_VEL
LIN {X 0,Y 153.024,Z 1121.29,A -85,B 0,C 180,E1 198.66,E2 198.66} C_VEL
LIN {X 0,Y 171.132,Z 1108.899,A -85,B 0,C 180,E1 194.099,E2 194.099} C_VEL
LIN {X 0,Y 188.528,Z 1095.546,A -85,B 0,C 180,E1 190.697,E2 190.697} C_VEL
LIN {X 0,Y 205.005,Z 1081.085,A -85,B 0,C 180,E1 188.075,E2 188.075} C_VEL
LIN {X 0,Y 221.634,Z 1064.593,A -85,B 0,C 180,E1 185.874,E2 185.874} C_VEL
LIN {X 0,Y 236.061,Z 1048.359,A -85,B 0,C 180,E1 184.245,E2 184.245} C_VEL
LIN {X 0,Y 249.291,Z 1031.242,A -85,B 0,C 180,E1 182.928,E2 182.928} C_VEL
LIN {X 0,Y 262.093,Z 1012.389,A -85,B 0,C 180,E1 181.797,E2 181.797} C_VEL
LIN {X 0,Y 273.495,Z 992.627,A -85,B 0,C 180,E1 180.884,E2 180.884} C_VEL
LIN {X 0,Y 283.962,Z 971.09,A -85,B 0,C 180,E1 180.115,E2 180.115} C_VEL
LIN {X 0,Y 292.455,Z 950.008,A -85,B 0,C 180,E1 179.537,E2 179.537} C_VEL
LIN {X 0,Y 299.278,Z 928.393,A -85,B 0,C 180,E1 179.096,E2 179.096} C_VEL
LIN {X 0,Y 305.004,Z 904.257,A -85,B 0,C 180,E1 178.709,E2 178.709} C_VEL
LIN {X 0,Y 308.72,Z 881.069,A -85,B 0,C 180,E1 178.373,E2 178.373} C_VEL
LIN {X 0,Y 312.825,Z 847.49,A -85,B 0,C 180,E1 177.888,E2 177.888} C_VEL
LIN {X 0,Y 306.475,Z 896.534,A -85,B 0,C 180,E1 177.22,E2 177.22} C_VEL
LIN {X 0,Y 301.683,Z 919.27,A -85,B 0,C 180,E1 176.895,E2 176.895} C_VEL
LIN {X 0,Y 295.013,Z 942.383,A -85,B 0,C 180,E1 176.492,E2 176.492} C_VEL
LIN {X 0,Y 287.168,Z 963.756,A -85,B 0,C 180,E1 175.978,E2 175.978} C_VEL
LIN {X 0,Y 277.884,Z 984.066,A -85,B 0,C 180,E1 175.332,E2 175.332} C_VEL
LIN {X 0,Y 266.213,Z 1005.481,A -85,B 0,C 180,E1 174.446,E2 174.446} C_VEL
LIN {X 0,Y 254.137,Z 1024.369,A -85,B 0,C 180,E1 173.427,E2 173.427} C_VEL
LIN {X 0,Y 240.715,Z 1042.262,A -85,B 0,C 180,E1 172.165,E2 172.165} C_VEL
LIN {X 0,Y 225.932,Z 1059.5,A -85,B 0,C 180,E1 170.575,E2 170.575} C_VEL
LIN {X 0,Y 211.052,Z 1074.676,A -85,B 0,C 180,E1 168.716,E2 168.716} C_VEL
LIN {X 0,Y 194.525,Z 1089.413,A -85,B 0,C 180,E1 166.279,E2 166.279} C_VEL
LIN {X 0,Y 178.423,Z 1102.16,A -85,B 0,C 180,E1 163.388,E2 163.388} C_VEL
LIN {X 0,Y 162.003,Z 1113.518,A -85,B 0,C 180,E1 159.739,E2 159.739} C_VEL
LIN {X 0,Y 143.987,Z 1124.552,A -85,B 0,C 180,E1 154.52,E2 154.52} C_VEL
LIN {X 0,Y 128.146,Z 1133.209,A -85,B 0,C 180,E1 148.263,E2 148.263} C_VEL
LIN {X 0,Y 113.507,Z 1140.282,A -85,B 0,C 180,E1 140.029,E2 140.029} C_VEL
LIN {X 0,Y 101.15,Z 1145.862,A -85,B 0,C 180,E1 129.245,E2 129.245} C_VEL
LIN {X 0,Y 92.98,Z 1149.59,A -85,B 0,C 180,E1 116.803,E2 116.803} C_VEL
LIN {X 0,Y 89.012,Z 1151.532,A -85,B 0,C 180,E1 103.644,E2 103.644} C_VEL
LIN {X 0,Y 88.141,Z 1152.161,A -85,B 0,C 180,E1 93.251,E2 93.251} C_VEL
LIN {X 0,Y 88.196,Z 1152.108,A -85,B 0,C 180,E1 84.796,E2 84.796} C_VEL
LIN {X 0,Y 89.463,Z 1151.307,A -85,B 0,C 180,E1 73.775,E2 73.775} C_VEL
LIN {X 0,Y 94.456,Z 1148.878,A -85,B 0,C 180,E1 60.164,E2 60.164} C_VEL
LIN {X 0,Y 103.483,Z 1144.944,A -85,B 0,C 180,E1 48.188,E2 48.188} C_VEL
LIN {X 0,Y 115.922,Z 1139.213,A -85,B 0,C 180,E1 38.288,E2 38.288} C_VEL
LIN {X 0,Y 131.7,Z 1131.39,A -85,B 0,C 180,E1 30.061,E2 30.061} C_VEL
LIN {X 0,Y 132.65,Z 1130.854,A -85,B 0,C 180,E1 29.586,E2 29.586} C_VEL
LIN {X 0,Y 117.206,Z 1133.126,A -85,B 0,C 180,E1 15.843,E2 15.843} C_VEL
LIN {X 0,Y 113.08,Z 1136.318,A -85,B 0,C 180,E1 -13.289,E2 -13.289} C_VEL
LIN {X 0,Y 123.995,Z 1137.416,A -85,B 0,C 180,E1 -27.362,E2 -27.362} C_VEL
LIN {X 0,Y 125.777,Z 1137.548,A -85,B 0,C 180,E1 -28.88,E2 -28.88} C_VEL
LIN {X 0,Y 111.749,Z 1144.875,A -85,B 0,C 180,E1 -37.219,E2 -37.219} C_VEL
LIN {X 0,Y 99.616,Z 1151.049,A -85,B 0,C 180,E1 -48.513,E2 -48.513} C_VEL
LIN {X 0,Y 92.15,Z 1155.09,A -85,B 0,C 180,E1 -60.773,E2 -60.773} C_VEL
LIN {X 0,Y 88.554,Z 1157.584,A -85,B 0,C 180,E1 -74.277,E2 -74.277} C_VEL
LIN {X 0,Y 88.045,Z 1158.458,A -85,B 0,C 180,E1 -84.134,E2 -84.134} C_VEL
LIN {X 0,Y 88.079,Z 1158.608,A -85,B 0,C 180,E1 -91.951,E2 -91.951} C_VEL
LIN {X 0,Y 88.148,Z 1158.098,A -85,B 0,C 180,E1 -101.118,E2 -101.118} C_VEL
LIN {X 0,Y 89.959,Z 1156.419,A -85,B 0,C 180,E1 -112.893,E2 -112.893} C_VEL
LIN {X 0,Y 95.586,Z 1153.178,A -85,B 0,C 180,E1 -125.858,E2 -125.858} C_VEL
LIN {X 0,Y 105.523,Z 1147.983,A -85,B 0,C 180,E1 -137.723,E2 -137.723} C_VEL
LIN {X 0,Y 119.416,Z 1140.838,A -85,B 0,C 180,E1 -147.743,E2 -147.743} C_VEL
LIN {X 0,Y 121.303,Z 1139.817,A -85,B 0,C 180,E1 -148.805,E2 -148.805} C_VEL
LIN {X 0,Y 125.437,Z 1137.352,A -85,B 0,C 180,E1 -151.623,E2 -151.623} C_VEL
LIN {X 0,Y 135.131,Z 1130.267,A -85,B 0,C 180,E1 -159.346,E2 -159.346} C_VEL
LIN {X 0,Y 139.425,Z 1127.608,A -85,B 0,C 180,E1 -161.172,E2 -161.172} C_VEL
LIN {X 0,Y 158.472,Z 1115.923,A -85,B 0,C 180,E1 -166.324,E2 -166.324} C_VEL
LIN {X 0,Y 175.716,Z 1104.021,A -85,B 0,C 180,E1 -169.869,E2 -169.869} C_VEL
LIN {X 0,Y 192.556,Z 1090.71,A -85,B 0,C 180,E1 -172.651,E2 -172.651} C_VEL
LIN {X 0,Y 209.777,Z 1075.38,A -85,B 0,C 180,E1 -174.976,E2 -174.976} C_VEL
LIN {X 0,Y 225.334,Z 1059.588,A -85,B 0,C 180,E1 -176.74,E2 -176.74} C_VEL
LIN {X 0,Y 240.455,Z 1041.958,A -85,B 0,C 180,E1 -178.218,E2 -178.218} C_VEL
LIN {X 0,Y 253.98,Z 1023.943,A -85,B 0,C 180,E1 -179.374,E2 -179.374} C_VEL
LIN {X 0,Y 265.967,Z 1005.325,A -85,B 0,C 180,E1 -180.292,E2 -180.292} C_VEL
LIN {X 0,Y 277.513,Z 984.315,A -85,B 0,C 180,E1 -181.097,E2 -181.097} C_VEL
LIN {X 0,Y 286.568,Z 964.747,A -85,B 0,C 180,E1 -181.683,E2 -181.683} C_VEL
LIN {X 0,Y 292.783,Z 948.706,A -85,B 0,C 180,E1 -182.07,E2 -182.07} C_VEL
LIN {X 0,Y 284.248,Z 970.008,A -85,B 0,C 180,E1 -182.576,E2 -182.576} C_VEL
LIN {X 0,Y 274.395,Z 990.44,A -85,B 0,C 180,E1 -183.219,E2 -183.219} C_VEL
LIN {X 0,Y 263.598,Z 1009.175,A -85,B 0,C 180,E1 -183.974,E2 -183.974} C_VEL
LIN {X 0,Y 250.419,Z 1028.778,A -85,B 0,C 180,E1 -185.001,E2 -185.001} C_VEL
LIN {X 0,Y 236.85,Z 1046.264,A -85,B 0,C 180,E1 -186.194,E2 -186.194} C_VEL
LIN {X 0,Y 221.964,Z 1062.776,A -85,B 0,C 180,E1 -187.685,E2 -187.685} C_VEL
LIN {X 0,Y 205.842,Z 1078.49,A -85,B 0,C 180,E1 -189.579,E2 -189.579} C_VEL
LIN {X 0,Y 189.058,Z 1092.772,A -85,B 0,C 180,E1 -191.93,E2 -191.93} C_VEL
LIN {X 0,Y 171.758,Z 1105.592,A -85,B 0,C 180,E1 -194.908,E2 -194.908} C_VEL
LIN {X 0,Y 154.153,Z 1117.099,A -85,B 0,C 180,E1 -198.741,E2 -198.741} C_VEL
LIN {X 0,Y 137.385,Z 1126.647,A -85,B 0,C 180,E1 -203.508,E2 -203.508} C_VEL
LIN {X 0,Y 120.293,Z 1135.219,A -85,B 0,C 180,E1 -210.182,E2 -210.182} C_VEL
LIN {X 0,Y 105.219,Z 1142.008,A -85,B 0,C 180,E1 -218.811,E2 -218.811} C_VEL
LIN {X 0,Y 92.996,Z 1146.948,A -85,B 0,C 180,E1 -229.827,E2 -229.827} C_VEL
LIN {X 0,Y 84.335,Z 1150.422,A -85,B 0,C 180,E1 -243.981,E2 -243.981} C_VEL
LIN {X 0,Y 80.859,Z 1152.013,A -85,B 0,C 180,E1 -257.14,E2 -257.14} C_VEL
LIN {X 0,Y 80.129,Z 1152.538,A -85,B 0,C 180,E1 -269.285,E2 -269.285} C_VEL
LIN {X 0,Y 80.583,Z 1152.225,A -85,B 0,C 180,E1 -280.726,E2 -280.726} C_VEL
LIN {X 0,Y 83.781,Z 1150.674,A -85,B 0,C 180,E1 -294.69,E2 -294.69} C_VEL
LIN {X 0,Y 91.566,Z 1147.607,A -85,B 0,C 180,E1 -308.493,E2 -308.493} C_VEL
LIN {X 0,Y 103.3,Z 1142.822,A -85,B 0,C 180,E1 -319.877,E2 -319.877} C_VEL
LIN {X 0,Y 118.765,Z 1136.017,A -85,B 0,C 180,E1 -329.174,E2 -329.174} C_VEL
LIN {X 0,Y 122.495,Z 1134.242,A -85,B 0,C 180,E1 -331.053,E2 -331.053} C_VEL
LIN {X 0,Y 104.946,Z 1136.997,A -85,B 0,C 180,E1 -352.884,E2 -352.884} C_VEL
LIN {X 0,Y 107.563,Z 1139.292,A -85,B 0,C 180,E1 -377.862,E2 -377.862} C_VEL
LIN {X 0,Y 116.152,Z 1140.097,A -85,B 0,C 180,E1 -388.208,E2 -388.208} C_VEL
LIN {X 0,Y 100.634,Z 1147.483,A -85,B 0,C 180,E1 -398.287,E2 -398.287} C_VEL
LIN {X 0,Y 89.403,Z 1152.714,A -85,B 0,C 180,E1 -410.396,E2 -410.396} C_VEL
LIN {X 0,Y 82.671,Z 1156.019,A -85,B 0,C 180,E1 -424.189,E2 -424.189} C_VEL
LIN {X 0,Y 80.259,Z 1157.741,A -85,B 0,C 180,E1 -437.041,E2 -437.041} C_VEL
LIN {X 0,Y 80.072,Z 1158.303,A -85,B 0,C 180,E1 -447.334,E2 -447.334} C_VEL
LIN {X 0,Y 80.051,Z 1158.215,A -85,B 0,C 180,E1 -455.016,E2 -455.016} C_VEL
LIN {X 0,Y 80.462,Z 1157.502,A -85,B 0,C 180,E1 -465.127,E2 -465.127} C_VEL
LIN {X 0,Y 83.883,Z 1155.377,A -85,B 0,C 180,E1 -479.256,E2 -479.256} C_VEL
LIN {X 0,Y 92.081,Z 1151.363,A -85,B 0,C 180,E1 -493.164,E2 -493.164} C_VEL
LIN {X 0,Y 104.308,Z 1145.776,A -85,B 0,C 180,E1 -504.566,E2 -504.566} C_VEL
LIN {X 0,Y 119.561,Z 1138.326,A -85,B 0,C 180,E1 -513.485,E2 -513.485} C_VEL
LIN {X 0,Y 137.007,Z 1128.983,A -85,B 0,C 180,E1 -520.386,E2 -520.386} C_VEL
LIN {X 0,Y 139.425,Z 1127.608,A -85,B 0,C 180,E1 -521.172,E2 -521.172} C_VEL
LIN {X 0,Y 144.476,Z 1124.477,A -85,B 0,C 180,E1 -523.187,E2 -523.187} C_VEL
LIN {X 0,Y 155.852,Z 1116.323,A -85,B 0,C 180,E1 -528.71,E2 -528.71} C_VEL
LIN {X 0,Y 161.283,Z 1112.683,A -85,B 0,C 180,E1 -530.232,E2 -530.232} C_VEL
LIN {X 0,Y 179.185,Z 1100.13,A -85,B 0,C 180,E1 -533.339,E2 -533.339} C_VEL
LIN {X 0,Y 196.514,Z 1086.422,A -85,B 0,C 180,E1 -535.75,E2 -535.75} C_VEL
LIN {X 0,Y 213.147,Z 1071.259,A -85,B 0,C 180,E1 -537.667,E2 -537.667} C_VEL
LIN {X 0,Y 229.986,Z 1053.729,A -85,B 0,C 180,E1 -539.3,E2 -539.3} C_VEL
LIN {X 0,Y 244.476,Z 1036.454,A -85,B 0,C 180,E1 -540.511,E2 -540.511} C_VEL
LIN {X 0,Y 258.055,Z 1017.531,A -85,B 0,C 180,E1 -541.52,E2 -541.52} C_VEL
LIN {X 0,Y 266.007,Z 1005.04,A -85,B 0,C 180,E1 -542.05,E2 -542.05} C_VEL
LIN {X 0,Y 253.786,Z 1023.813,A -85,B 0,C 180,E1 -542.879,E2 -542.879} C_VEL
LIN {X 0,Y 240.52,Z 1041.244,A -85,B 0,C 180,E1 -543.885,E2 -543.885} C_VEL
LIN {X 0,Y 225.88,Z 1058.124,A -85,B 0,C 180,E1 -545.148,E2 -545.148} C_VEL
LIN {X 0,Y 210.407,Z 1073.545,A -85,B 0,C 180,E1 -546.698,E2 -546.698} C_VEL
LIN {X 0,Y 193.216,Z 1088.547,A -85,B 0,C 180,E1 -548.737,E2 -548.737} C_VEL
LIN {X 0,Y 175.39,Z 1102.152,A -85,B 0,C 180,E1 -551.322,E2 -551.322} C_VEL
LIN {X 0,Y 157.091,Z 1114.141,A -85,B 0,C 180,E1 -554.657,E2 -554.657} C_VEL
LIN {X 0,Y 138.595,Z 1124.715,A -85,B 0,C 180,E1 -559.078,E2 -559.078} C_VEL
LIN {X 0,Y 121.129,Z 1133.441,A -85,B 0,C 180,E1 -564.77,E2 -564.77} C_VEL
LIN {X 0,Y 104.449,Z 1140.59,A -85,B 0,C 180,E1 -572.606,E2 -572.606} C_VEL
LIN {X 0,Y 89.068,Z 1146.464,A -85,B 0,C 180,E1 -584.109,E2 -584.109} C_VEL
LIN {X 0,Y 78.821,Z 1150.173,A -85,B 0,C 180,E1 -597.806,E2 -597.806} C_VEL
LIN {X 0,Y 73.421,Z 1152.119,A -85,B 0,C 180,E1 -613.383,E2 -613.383} C_VEL
LIN {X 0,Y 72.164,Z 1152.744,A -85,B 0,C 180,E1 -626.048,E2 -626.048} C_VEL
LIN {X 0,Y 72.213,Z 1152.71,A -85,B 0,C 180,E1 -635.562,E2 -635.562} C_VEL
LIN {X 0,Y 73.768,Z 1151.999,A -85,B 0,C 180,E1 -648.41,E2 -648.41} C_VEL
LIN {X 0,Y 80.318,Z 1149.621,A -85,B 0,C 180,E1 -664.935,E2 -664.935} C_VEL
LIN {X 0,Y 91.339,Z 1145.733,A -85,B 0,C 180,E1 -678.106,E2 -678.106} C_VEL
LIN {X 0,Y 105.821,Z 1140.098,A -85,B 0,C 180,E1 -688.253,E2 -688.253} C_VEL
LIN {X 0,Y 112.496,Z 1137.305,A -85,B 0,C 180,E1 -691.765,E2 -691.765} C_VEL
LIN {X 0,Y 96.754,Z 1139.876,A -85,B 0,C 180,E1 -715.256,E2 -715.256} C_VEL
LIN {X 0,Y 99.765,Z 1141.768,A -85,B 0,C 180,E1 -738.099,E2 -738.099} C_VEL
LIN {X 0,Y 106.63,Z 1142.455,A -85,B 0,C 180,E1 -747.351,E2 -747.351} C_VEL
LIN {X 0,Y 92.506,Z 1148.516,A -85,B 0,C 180,E1 -756.885,E2 -756.885} C_VEL
LIN {X 0,Y 80.474,Z 1153.463,A -85,B 0,C 180,E1 -770.679,E2 -770.679} C_VEL
LIN {X 0,Y 74.166,Z 1156.336,A -85,B 0,C 180,E1 -785.296,E2 -785.296} C_VEL
LIN {X 0,Y 72.1,Z 1157.79,A -85,B 0,C 180,E1 -800.421,E2 -800.421} C_VEL
LIN {X 0,Y 72.108,Z 1158.093,A -85,B 0,C 180,E1 -810,E2 -810} C_VEL
LIN {X 0,Y 72.121,Z 1157.757,A -85,B 0,C 180,E1 -820.383,E2 -820.383} C_VEL
LIN {X 0,Y 74.605,Z 1156.067,A -85,B 0,C 180,E1 -836.249,E2 -836.249} C_VEL
LIN {X 0,Y 81.329,Z 1153.089,A -85,B 0,C 180,E1 -850.661,E2 -850.661} C_VEL
LIN {X 0,Y 93.751,Z 1147.934,A -85,B 0,C 180,E1 -864.149,E2 -864.149} C_VEL
LIN {X 0,Y 109.079,Z 1141.32,A -85,B 0,C 180,E1 -873.936,E2 -873.936} C_VEL
LIN {X 0,Y 126.679,Z 1132.763,A -85,B 0,C 180,E1 -881.288,E2 -881.288} C_VEL
LIN {X 0,Y 144.914,Z 1122.776,A -85,B 0,C 180,E1 -886.621,E2 -886.621} C_VEL
LIN {X 0,Y 161.283,Z 1112.683,A -85,B 0,C 180,E1 -890.232,E2 -890.232} C_VEL
LIN {X 0,Y 166.782,Z 1108.973,A -85,B 0,C 180,E1 -891.645,E2 -891.645} C_VEL
LIN {X 0,Y 179.325,Z 1099.368,A -85,B 0,C 180,E1 -895.778,E2 -895.778} C_VEL
LIN {X 0,Y 184.832,Z 1095.073,A -85,B 0,C 180,E1 -896.842,E2 -896.842} C_VEL
LIN {X 0,Y 202.515,Z 1080.487,A -85,B 0,C 180,E1 -898.869,E2 -898.869} C_VEL
LIN {X 0,Y 219.979,Z 1064.001,A -85,B 0,C 180,E1 -900.53,E2 -900.53} C_VEL
LIN {X 0,Y 235.582,Z 1047.144,A -85,B 0,C 180,E1 -901.783,E2 -901.783} C_VEL
LIN {X 0,Y 238.872,Z 1043.142,A -85,B 0,C 180,E1 -902.056,E2 -902.056} C_VEL
LIN {X 0,Y 222.84,Z 1060.986,A -85,B 0,C 180,E1 -903.303,E2 -903.303} C_VEL
LIN {X 0,Y 206.692,Z 1076.629,A -85,B 0,C 180,E1 -904.786,E2 -904.786} C_VEL
LIN {X 0,Y 189.259,Z 1091.151,A -85,B 0,C 180,E1 -906.679,E2 -906.679} C_VEL
LIN {X 0,Y 170.186,Z 1104.971,A -85,B 0,C 180,E1 -909.242,E2 -909.242} C_VEL
LIN {X 0,Y 151.538,Z 1116.691,A -85,B 0,C 180,E1 -912.441,E2 -912.441} C_VEL
LIN {X 0,Y 132.592,Z 1126.81,A -85,B 0,C 180,E1 -916.725,E2 -916.725} C_VEL
LIN {X 0,Y 113.212,Z 1135.711,A -85,B 0,C 180,E1 -922.869,E2 -922.869} C_VEL
LIN {X 0,Y 96.537,Z 1142.35,A -85,B 0,C 180,E1 -930.722,E2 -930.722} C_VEL
LIN {X 0,Y 81.785,Z 1147.347,A -85,B 0,C 180,E1 -941.776,E2 -941.776} C_VEL
LIN {X 0,Y 70.096,Z 1151.013,A -85,B 0,C 180,E1 -958.145,E2 -958.145} C_VEL
LIN {X 0,Y 65.242,Z 1152.6,A -85,B 0,C 180,E1 -973.987,E2 -973.987} C_VEL
LIN {X 0,Y 64.14,Z 1153.098,A -85,B 0,C 180,E1 -988.214,E2 -988.214} C_VEL
LIN {X 0,Y 64.549,Z 1152.904,A -85,B 0,C 180,E1 -1000.713,E2 -1000.713} C_VEL
LIN {X 0,Y 68.692,Z 1151.475,A -85,B 0,C 180,E1 -1018.708,E2 -1018.708} C_VEL
LIN {X 0,Y 78.32,Z 1148.554,A -85,B 0,C 180,E1 -1034.6,E2 -1034.6} C_VEL
LIN {X 0,Y 92.165,Z 1143.902,A -85,B 0,C 180,E1 -1046.652,E2 -1046.652} C_VEL
LIN {X 0,Y 102.464,Z 1140.09,A -85,B 0,C 180,E1 -1052.7,E2 -1052.7} C_VEL
LIN {X 0,Y 89.015,Z 1142.242,A -85,B 0,C 180,E1 -1075.489,E2 -1075.489} C_VEL
LIN {X 0,Y 92.204,Z 1144.056,A -85,B 0,C 180,E1 -1098.983,E2 -1098.983} C_VEL
LIN {X 0,Y 97.072,Z 1144.592,A -85,B 0,C 180,E1 -1106.347,E2 -1106.347} C_VEL
LIN {X 0,Y 81.744,Z 1150.428,A -85,B 0,C 180,E1 -1117.701,E2 -1117.701} C_VEL
LIN {X 0,Y 70.717,Z 1154.529,A -85,B 0,C 180,E1 -1132.557,E2 -1132.557} C_VEL
LIN {X 0,Y 65,Z 1156.847,A -85,B 0,C 180,E1 -1150.22,E2 -1150.22} C_VEL
LIN {X 0,Y 64.058,Z 1157.635,A -85,B 0,C 180,E1 -1163.727,E2 -1163.727} C_VEL
LIN {X 0,Y 64.08,Z 1157.734,A -85,B 0,C 180,E1 -1172.683,E2 -1172.683} C_VEL
LIN {X 0,Y 64.431,Z 1157.212,A -85,B 0,C 180,E1 -1185.296,E2 -1185.296} C_VEL
LIN {X 0,Y 68.216,Z 1155.398,A -85,B 0,C 180,E1 -1201.848,E2 -1201.848} C_VEL
LIN {X 0,Y 77.865,Z 1151.848,A -85,B 0,C 180,E1 -1218.14,E2 -1218.14} C_VEL
LIN {X 0,Y 91.209,Z 1146.827,A -85,B 0,C 180,E1 -1230,E2 -1230} C_VEL
LIN {X 0,Y 108.912,Z 1139.545,A -85,B 0,C 180,E1 -1239.456,E2 -1239.456} C_VEL
LIN {X 0,Y 127.553,Z 1130.871,A -85,B 0,C 180,E1 -1245.937,E2 -1245.937} C_VEL
LIN {X 0,Y 146.281,Z 1120.705,A -85,B 0,C 180,E1 -1250.559,E2 -1250.559} C_VEL
LIN {X 0,Y 165.842,Z 1108.581,A -85,B 0,C 180,E1 -1254.146,E2 -1254.146} C_VEL
LIN {X 0,Y 184.268,Z 1095.51,A -85,B 0,C 180,E1 -1256.77,E2 -1256.77} C_VEL
LIN {X 0,Y 184.832,Z 1095.073,A -85,B 0,C 180,E1 -1256.842,E2 -1256.842} C_VEL
LIN {X 0,Y 190.354,Z 1090.681,A -85,B 0,C 180,E1 -1257.838,E2 -1257.838} C_VEL
LIN {X 0,Y 203.23,Z 1079.653,A -85,B 0,C 180,E1 -1261.001,E2 -1261.001} C_VEL
LIN {X 0,Y 208.593,Z 1074.759,A -85,B 0,C 180,E1 -1261.756,E2 -1261.756} C_VEL
LIN {X 0,Y 211.858,Z 1071.721,A -85,B 0,C 180,E1 -1262.054,E2 -1262.054} C_VEL
LIN {X 0,Y 195.344,Z 1086.152,A -85,B 0,C 180,E1 -1263.533,E2 -1263.533} C_VEL
LIN {X 0,Y 177.77,Z 1099.354,A -85,B 0,C 180,E1 -1265.42,E2 -1265.42} C_VEL
LIN {X 0,Y 158.525,Z 1111.945,A -85,B 0,C 180,E1 -1268.011,E2 -1268.011} C_VEL
LIN {X 0,Y 139.686,Z 1122.551,A -85,B 0,C 180,E1 -1271.294,E2 -1271.294} C_VEL
LIN {X 0,Y 120.536,Z 1131.683,A -85,B 0,C 180,E1 -1275.797,E2 -1275.797} C_VEL
LIN {X 0,Y 101.531,Z 1139.431,A -85,B 0,C 180,E1 -1282.226,E2 -1282.226} C_VEL
LIN {X 0,Y 84.983,Z 1145.105,A -85,B 0,C 180,E1 -1290.81,E2 -1290.81} C_VEL
LIN {X 0,Y 69.824,Z 1149.558,A -85,B 0,C 180,E1 -1304.276,E2 -1304.276} C_VEL
LIN {X 0,Y 59.992,Z 1152.264,A -85,B 0,C 180,E1 -1322.182,E2 -1322.182} C_VEL
LIN {X 0,Y 56.407,Z 1153.246,A -85,B 0,C 180,E1 -1340.82,E2 -1340.82} C_VEL
LIN {X 0,Y 56.154,Z 1153.374,A -85,B 0,C 180,E1 -1353.062,E2 -1353.062} C_VEL
LIN {X 0,Y 57.694,Z 1152.852,A -85,B 0,C 180,E1 -1369.225,E2 -1369.225} C_VEL
LIN {X 0,Y 64.176,Z 1151.132,A -85,B 0,C 180,E1 -1387.418,E2 -1387.418} C_VEL
LIN {X 0,Y 77.233,Z 1147.498,A -85,B 0,C 180,E1 -1403.448,E2 -1403.448} C_VEL
LIN {X 0,Y 92.428,Z 1142.769,A -85,B 0,C 180,E1 -1413.669,E2 -1413.669} C_VEL
LIN {X 0,Y 82.633,Z 1145.855,A -85,B 0,C 180,E1 -1455.436,E2 -1455.436} C_VEL
LIN {X 0,Y 87.536,Z 1146.501,A -85,B 0,C 180,E1 -1465.11,E2 -1465.11} C_VEL
LIN {X 0,Y 71.954,Z 1151.807,A -85,B 0,C 180,E1 -1477.621,E2 -1477.621} C_VEL
LIN {X 0,Y 61.36,Z 1155.12,A -85,B 0,C 180,E1 -1494.082,E2 -1494.082} C_VEL
LIN {X 0,Y 56.621,Z 1156.93,A -85,B 0,C 180,E1 -1512.53,E2 -1512.53} C_VEL
LIN {X 0,Y 56.078,Z 1157.448,A -85,B 0,C 180,E1 -1526.934,E2 -1526.934} C_VEL
LIN {X 0,Y 56.061,Z 1157.365,A -85,B 0,C 180,E1 -1536.143,E2 -1536.143} C_VEL
LIN {X 0,Y 57.196,Z 1156.613,A -85,B 0,C 180,E1 -1551.537,E2 -1551.537} C_VEL
LIN {X 0,Y 63.876,Z 1154.351,A -85,B 0,C 180,E1 -1571.104,E2 -1571.104} C_VEL
LIN {X 0,Y 76.455,Z 1150.234,A -85,B 0,C 180,E1 -1586.822,E2 -1586.822} C_VEL
LIN {X 0,Y 93.648,Z 1144.221,A -85,B 0,C 180,E1 -1598.261,E2 -1598.261} C_VEL
LIN {X 0,Y 111.517,Z 1137.036,A -85,B 0,C 180,E1 -1605.54,E2 -1605.54} C_VEL
LIN {X 0,Y 130.649,Z 1128.081,A -85,B 0,C 180,E1 -1610.839,E2 -1610.839} C_VEL
LIN {X 0,Y 149.725,Z 1117.85,A -85,B 0,C 180,E1 -1614.637,E2 -1614.637} C_VEL
LIN {X 0,Y 169.129,Z 1105.661,A -85,B 0,C 180,E1 -1617.571,E2 -1617.571} C_VEL
LIN {X 0,Y 187.975,Z 1092.062,A -85,B 0,C 180,E1 -1619.807,E2 -1619.807} C_VEL
LIN {X 0,Y 206.046,Z 1077.125,A -85,B 0,C 180,E1 -1621.536,E2 -1621.536} C_VEL
LIN {X 0,Y 208.593,Z 1074.759,A -85,B 0,C 180,E1 -1621.756,E2 -1621.756} C_VEL
LIN {X 0,Y 207.265,Z 1075.995,A -85,B 0,C 180,E1 -1622.008,E2 -1622.008} C_VEL
LIN {X 0,Y 199.98,Z 1082.238,A -85,B 0,C 180,E1 -1622.173,E2 -1622.173} C_VEL
LIN {X 0,Y 185.472,Z 1093.808,A -85,B 0,C 180,E1 -1621.821,E2 -1621.821} C_VEL
LIN {X 0,Y 175.426,Z 1100.99,A -85,B 0,C 180,E1 -1621.108,E2 -1621.108} C_VEL
LIN {X 0,Y 156.012,Z 1113.479,A -85,B 0,C 180,E1 -1618.815,E2 -1618.815} C_VEL
LIN {X 0,Y 136.352,Z 1124.46,A -85,B 0,C 180,E1 -1615.775,E2 -1615.775} C_VEL
LIN {X 0,Y 116.25,Z 1133.927,A -85,B 0,C 180,E1 -1611.538,E2 -1611.538} C_VEL
LIN {X 0,Y 95.242,Z 1142.334,A -85,B 0,C 180,E1 -1604.977,E2 -1604.977} C_VEL
LIN {X 0,Y 76.819,Z 1148.61,A -85,B 0,C 180,E1 -1595.659,E2 -1595.659} C_VEL
LIN {X 0,Y 61.322,Z 1153.038,A -85,B 0,C 180,E1 -1581.503,E2 -1581.503} C_VEL
LIN {X 0,Y 51.021,Z 1155.932,A -85,B 0,C 180,E1 -1560.632,E2 -1560.632} C_VEL
LIN {X 0,Y 48.134,Z 1156.989,A -85,B 0,C 180,E1 -1540.775,E2 -1540.775} C_VEL
LIN {X 0,Y 48.103,Z 1157.206,A -85,B 0,C 180,E1 -1528.809,E2 -1528.809} C_VEL
LIN {X 0,Y 48.498,Z 1156.847,A -85,B 0,C 180,E1 -1513.224,E2 -1513.224} C_VEL
LIN {X 0,Y 53.993,Z 1155.068,A -85,B 0,C 180,E1 -1490.977,E2 -1490.977} C_VEL
LIN {X 0,Y 66.247,Z 1151.77,A -85,B 0,C 180,E1 -1472.909,E2 -1472.909} C_VEL
LIN {X 0,Y 78.116,Z 1148.209,A -85,B 0,C 180,E1 -1463.376,E2 -1463.376} C_VEL
LIN {X 0,Y 73.205,Z 1146.584,A -85,B 0,C 180,E1 -1436.866,E2 -1436.866} C_VEL
LIN {X 0,Y 82.352,Z 1145.076,A -85,B 0,C 180,E1 -1414.966,E2 -1414.966} C_VEL
LIN {X 0,Y 64.997,Z 1149.749,A -85,B 0,C 180,E1 -1401.679,E2 -1401.679} C_VEL
LIN {X 0,Y 53.712,Z 1152.383,A -85,B 0,C 180,E1 -1383.949,E2 -1383.949} C_VEL
LIN {X 0,Y 48.596,Z 1153.526,A -85,B 0,C 180,E1 -1361.874,E2 -1361.874} C_VEL
LIN {X 0,Y 48.166,Z 1153.658,A -85,B 0,C 180,E1 -1346.43,E2 -1346.43} C_VEL
LIN {X 0,Y 50.151,Z 1153.126,A -85,B 0,C 180,E1 -1327.741,E2 -1327.741} C_VEL
LIN {X 0,Y 57.952,Z 1151.393,A -85,B 0,C 180,E1 -1307.711,E2 -1307.711} C_VEL
LIN {X 0,Y 72.661,Z 1147.747,A -85,B 0,C 180,E1 -1291.443,E2 -1291.443} C_VEL
LIN {X 0,Y 90.123,Z 1142.663,A -85,B 0,C 180,E1 -1281.263,E2 -1281.263} C_VEL
LIN {X 0,Y 109.414,Z 1135.735,A -85,B 0,C 180,E1 -1274.381,E2 -1274.381} C_VEL
LIN {X 0,Y 129.778,Z 1126.969,A -85,B 0,C 180,E1 -1269.543,E2 -1269.543} C_VEL
LIN {X 0,Y 148.874,Z 1117.304,A -85,B 0,C 180,E1 -1266.284,E2 -1266.284} C_VEL
LIN {X 0,Y 168.415,Z 1105.547,A -85,B 0,C 180,E1 -1263.745,E2 -1263.745} C_VEL
LIN {X 0,Y 184.799,Z 1094.307,A -85,B 0,C 180,E1 -1262.036,E2 -1262.036} C_VEL
LIN {X 0,Y 175.426,Z 1100.99,A -85,B 0,C 180,E1 -1261.108,E2 -1261.108} C_VEL
LIN {X 0,Y 169.96,Z 1104.731,A -85,B 0,C 180,E1 -1260.844,E2 -1260.844} C_VEL
LIN {X 0,Y 162.445,Z 1109.496,A -85,B 0,C 180,E1 -1261.214,E2 -1261.214} C_VEL
LIN {X 0,Y 145.165,Z 1119.172,A -85,B 0,C 180,E1 -1263.524,E2 -1263.524} C_VEL
LIN {X 0,Y 125.777,Z 1128.618,A -85,B 0,C 180,E1 -1266.441,E2 -1266.441} C_VEL
LIN {X 0,Y 105.795,Z 1136.722,A -85,B 0,C 180,E1 -1270.612,E2 -1270.612} C_VEL
LIN {X 0,Y 85.621,Z 1143.519,A -85,B 0,C 180,E1 -1276.976,E2 -1276.976} C_VEL
LIN {X 0,Y 67.156,Z 1148.44,A -85,B 0,C 180,E1 -1286.706,E2 -1286.706} C_VEL
LIN {X 0,Y 51.013,Z 1151.901,A -85,B 0,C 180,E1 -1303.515,E2 -1303.515} C_VEL
LIN {X 0,Y 42.206,Z 1153.545,A -85,B 0,C 180,E1 -1326.251,E2 -1326.251} C_VEL
LIN {X 0,Y 40.153,Z 1153.992,A -85,B 0,C 180,E1 -1348.573,E2 -1348.573} C_VEL
LIN {X 0,Y 41.269,Z 1153.762,A -85,B 0,C 180,E1 -1368.359,E2 -1368.359} C_VEL
LIN {X 0,Y 49.279,Z 1152.251,A -85,B 0,C 180,E1 -1393.619,E2 -1393.619} C_VEL
LIN {X 0,Y 64.077,Z 1149.267,A -85,B 0,C 180,E1 -1411.068,E2 -1411.068} C_VEL
LIN {X 0,Y 72.367,Z 1147.204,A -85,B 0,C 180,E1 -1416.87,E2 -1416.87} C_VEL
LIN {X 0,Y 68.75,Z 1149.672,A -85,B 0,C 180,E1 -1461.442,E2 -1461.442} C_VEL
LIN {X 0,Y 52.524,Z 1153.777,A -85,B 0,C 180,E1 -1476.915,E2 -1476.915} C_VEL
LIN {X 0,Y 42.712,Z 1155.955,A -85,B 0,C 180,E1 -1499.002,E2 -1499.002} C_VEL
LIN {X 0,Y 40.078,Z 1156.784,A -85,B 0,C 180,E1 -1521.391,E2 -1521.391} C_VEL
LIN {X 0,Y 40.086,Z 1156.885,A -85,B 0,C 180,E1 -1532.859,E2 -1532.859} C_VEL
LIN {X 0,Y 41.138,Z 1156.398,A -85,B 0,C 180,E1 -1552.885,E2 -1552.885} C_VEL
LIN {X 0,Y 48.396,Z 1154.62,A -85,B 0,C 180,E1 -1576.311,E2 -1576.311} C_VEL
LIN {X 0,Y 63.168,Z 1151.153,A -85,B 0,C 180,E1 -1594.452,E2 -1594.452} C_VEL
LIN {X 0,Y 81.597,Z 1145.91,A -85,B 0,C 180,E1 -1605.476,E2 -1605.476} C_VEL
LIN {X 0,Y 102.891,Z 1138.593,A -85,B 0,C 180,E1 -1612.744,E2 -1612.744} C_VEL
LIN {X 0,Y 124.113,Z 1129.814,A -85,B 0,C 180,E1 -1617.373,E2 -1617.373} C_VEL
LIN {X 0,Y 143.984,Z 1119.936,A -85,B 0,C 180,E1 -1620.422,E2 -1620.422} C_VEL
LIN {X 0,Y 157.499,Z 1112.328,A -85,B 0,C 180,E1 -1622.046,E2 -1622.046} C_VEL
LIN {X 0,Y 145.165,Z 1119.172,A -85,B 0,C 180,E1 -1623.524,E2 -1623.524} C_VEL
LIN {X 0,Y 138.312,Z 1122.72,A -85,B 0,C 180,E1 -1624.026,E2 -1624.026} C_VEL
LIN {X 0,Y 120.011,Z 1131.082,A -85,B 0,C 180,E1 -1623.958,E2 -1623.958} C_VEL
LIN {X 0,Y 112.958,Z 1133.927,A -85,B 0,C 180,E1 -1624.622,E2 -1624.622} C_VEL
LIN {X 0,Y 92.144,Z 1141.206,A -85,B 0,C 180,E1 -1629.088,E2 -1629.088} C_VEL
LIN {X 0,Y 71.463,Z 1147.031,A -85,B 0,C 180,E1 -1636.252,E2 -1636.252} C_VEL
LIN {X 0,Y 52.812,Z 1150.975,A -85,B 0,C 180,E1 -1648.253,E2 -1648.253} C_VEL
LIN {X 0,Y 37.479,Z 1153.466,A -85,B 0,C 180,E1 -1672.151,E2 -1672.151} C_VEL
LIN {X 0,Y 32.545,Z 1154.16,A -85,B 0,C 180,E1 -1697.582,E2 -1697.582} C_VEL
LIN {X 0,Y 32.204,Z 1154.247,A -85,B 0,C 180,E1 -1715.345,E2 -1715.345} C_VEL
LIN {X 0,Y 35.7,Z 1153.733,A -85,B 0,C 180,E1 -1742.151,E2 -1742.151} C_VEL
LIN {X 0,Y 47.163,Z 1152.016,A -85,B 0,C 180,E1 -1765.773,E2 -1765.773} C_VEL
LIN {X 0,Y 62.363,Z 1149.141,A -85,B 0,C 180,E1 -1779.074,E2 -1779.074} C_VEL
LIN {X 0,Y 59.331,Z 1151.07,A -85,B 0,C 180,E1 -1818.825,E2 -1818.825} C_VEL
LIN {X 0,Y 42.452,Z 1154.47,A -85,B 0,C 180,E1 -1836.793,E2 -1836.793} C_VEL
LIN {X 0,Y 33.011,Z 1156.287,A -85,B 0,C 180,E1 -1866.811,E2 -1866.811} C_VEL
LIN {X 0,Y 32.099,Z 1156.624,A -85,B 0,C 180,E1 -1888.215,E2 -1888.215} C_VEL
LIN {X 0,Y 32.253,Z 1156.429,A -85,B 0,C 180,E1 -1904.359,E2 -1904.359} C_VEL
LIN {X 0,Y 37.815,Z 1155.334,A -85,B 0,C 180,E1 -1933.429,E2 -1933.429} C_VEL
LIN {X 0,Y 52.606,Z 1152.433,A -85,B 0,C 180,E1 -1955.828,E2 -1955.828} C_VEL
LIN {X 0,Y 71.562,Z 1147.999,A -85,B 0,C 180,E1 -1967.968,E2 -1967.968} C_VEL
LIN {X 0,Y 92.325,Z 1141.724,A -85,B 0,C 180,E1 -1975.096,E2 -1975.096} C_VEL
LIN {X 0,Y 114.985,Z 1133.306,A -85,B 0,C 180,E1 -1979.849,E2 -1979.849} C_VEL
LIN {X 0,Y 129.693,Z 1126.847,A -85,B 0,C 180,E1 -1982.085,E2 -1982.085} C_VEL
LIN {X 0,Y 112.958,Z 1133.927,A -85,B 0,C 180,E1 -1984.622,E2 -1984.622} C_VEL
LIN {X 0,Y 105.838,Z 1136.671,A -85,B 0,C 180,E1 -1985.384,E2 -1985.384} C_VEL
LIN {X 0,Y 85.623,Z 1143.211,A -85,B 0,C 180,E1 -1985.742,E2 -1985.742} C_VEL
LIN {X 0,Y 79.349,Z 1144.875,A -85,B 0,C 180,E1 -1986.772,E2 -1986.772} C_VEL
LIN {X 0,Y 57.898,Z 1149.824,A -85,B 0,C 180,E1 -1994.743,E2 -1994.743} C_VEL
LIN {X 0,Y 39.159,Z 1152.812,A -85,B 0,C 180,E1 -2009.757,E2 -2009.757} C_VEL
LIN {X 0,Y 26.471,Z 1154.341,A -85,B 0,C 180,E1 -2040.592,E2 -2040.592} C_VEL
LIN {X 0,Y 24.164,Z 1154.58,A -85,B 0,C 180,E1 -2072.372,E2 -2072.372} C_VEL
LIN {X 0,Y 27.691,Z 1154.214,A -85,B 0,C 180,E1 -2105.292,E2 -2105.292} C_VEL
LIN {X 0,Y 40.696,Z 1152.63,A -85,B 0,C 180,E1 -2132.189,E2 -2132.189} C_VEL
LIN {X 0,Y 52.499,Z 1150.788,A -85,B 0,C 180,E1 -2142.255,E2 -2142.255} C_VEL
LIN {X 0,Y 50.33,Z 1152.061,A -85,B 0,C 180,E1 -2174.964,E2 -2174.964} C_VEL
LIN {X 0,Y 32.913,Z 1154.983,A -85,B 0,C 180,E1 -2195.248,E2 -2195.248} C_VEL
LIN {X 0,Y 24.48,Z 1156.139,A -85,B 0,C 180,E1 -2230.927,E2 -2230.927} C_VEL
LIN {X 0,Y 24.093,Z 1156.328,A -85,B 0,C 180,E1 -2252.378,E2 -2252.378} C_VEL
LIN {X 0,Y 26.843,Z 1155.803,A -85,B 0,C 180,E1 -2286.581,E2 -2286.581} C_VEL
LIN {X 0,Y 39.641,Z 1153.895,A -85,B 0,C 180,E1 -2315.233,E2 -2315.233} C_VEL
LIN {X 0,Y 59.822,Z 1150.108,A -85,B 0,C 180,E1 -2330.445,E2 -2330.445} C_VEL
LIN {X 0,Y 80.06,Z 1145.035,A -85,B 0,C 180,E1 -2337.59,E2 -2337.59} C_VEL
LIN {X 0,Y 101.555,Z 1138.182,A -85,B 0,C 180,E1 -2342.101,E2 -2342.101} C_VEL
LIN {X 0,Y 79.349,Z 1144.875,A -85,B 0,C 180,E1 -2346.772,E2 -2346.772} C_VEL
LIN {X 0,Y 72,Z 1146.774,A -85,B 0,C 180,E1 -2348.098,E2 -2348.098} C_VEL
LIN {X 0,Y 51.768,Z 1150.862,A -85,B 0,C 180,E1 -2349.503,E2 -2349.503} C_VEL
LIN {X 0,Y 44.918,Z 1151.957,A -85,B 0,C 180,E1 -2351.846,E2 -2351.846} C_VEL
LIN {X 0,Y 25.834,Z 1154.117,A -85,B 0,C 180,E1 -2371.627,E2 -2371.627} C_VEL
LIN {X 0,Y 16.92,Z 1154.763,A -85,B 0,C 180,E1 -2409.234,E2 -2409.234} C_VEL
LIN {X 0,Y 16.326,Z 1154.829,A -85,B 0,C 180,E1 -2440.588,E2 -2440.588} C_VEL
LIN {X 0,Y 23.766,Z 1154.308,A -85,B 0,C 180,E1 -2483.907,E2 -2483.907} C_VEL
LIN {X 0,Y 41.275,Z 1152.497,A -85,B 0,C 180,E1 -2505.977,E2 -2505.977} C_VEL
LIN {X 0,Y 42.949,Z 1152.305,A -85,B 0,C 180,E1 -2507.341,E2 -2507.341} C_VEL
LIN {X 0,Y 41.401,Z 1153.023,A -85,B 0,C 180,E1 -2529.668,E2 -2529.668} C_VEL
LIN {X 0,Y 23.556,Z 1155.216,A -85,B 0,C 180,E1 -2551.905,E2 -2551.905} C_VEL
LIN {X 0,Y 16.11,Z 1155.988,A -85,B 0,C 180,E1 -2599.268,E2 -2599.268} C_VEL
LIN {X 0,Y 16.08,Z 1156.01,A -85,B 0,C 180,E1 -2617.143,E2 -2617.143} C_VEL
LIN {X 0,Y 22.841,Z 1155.276,A -85,B 0,C 180,E1 -2666.274,E2 -2666.274} C_VEL
LIN {X 0,Y 39.702,Z 1153.22,A -85,B 0,C 180,E1 -2689.167,E2 -2689.167} C_VEL
LIN {X 0,Y 61.995,Z 1149.15,A -85,B 0,C 180,E1 -2699.397,E2 -2699.397} C_VEL
LIN {X 0,Y 72.559,Z 1146.719,A -85,B 0,C 180,E1 -2702.085,E2 -2702.085} C_VEL
LIN {X 0,Y 50.161,Z 1151.114,A -85,B 0,C 180,E1 -2709.179,E2 -2709.179} C_VEL
LIN {X 0,Y 44.918,Z 1151.957,A -85,B 0,C 180,E1 -2711.846,E2 -2711.846} C_VEL
LIN {X 0,Y 37.611,Z 1153.008,A -85,B 0,C 180,E1 -2715.175,E2 -2715.175} C_VEL
LIN {X 0,Y 22.814,Z 1154.443,A -85,B 0,C 180,E1 -2720.618,E2 -2720.618} C_VEL
LIN {X 0,Y 13.456,Z 1154.961,A -85,B 0,C 180,E1 -2732.917,E2 -2732.917} C_VEL
LIN {X 0,Y 11.348,Z 1155.008,A -85,B 0,C 180,E1 -2741.454,E2 -2741.454} C_VEL
LIN {X 0,Y 8.34,Z 1155.141,A -85,B 0,C 180,E1 -2803.874,E2 -2803.874} C_VEL
LIN {X 0,Y 19.518,Z 1154.642,A -85,B 0,C 180,E1 -2862.091,E2 -2862.091} C_VEL
LIN {X 0,Y 33.669,Z 1153.491,A -85,B 0,C 180,E1 -2874.884,E2 -2874.884} C_VEL
LIN {X 0,Y 33.167,Z 1153.672,A -85,B 0,C 180,E1 -2881.369,E2 -2881.369} C_VEL
LIN {X 0,Y 13.44,Z 1155.428,A -85,B 0,C 180,E1 -2906.78,E2 -2906.78} C_VEL
LIN {X 0,Y 8.106,Z 1155.766,A -85,B 0,C 180,E1 -2969.999,E2 -2969.999} C_VEL
LIN {X 0,Y 16.811,Z 1155.206,A -85,B 0,C 180,E1 -3042.105,E2 -3042.105} C_VEL
LIN {X 0,Y 35.995,Z 1153.291,A -85,B 0,C 180,E1 -3060.008,E2 -3060.008} C_VEL
LIN {X 0,Y 41.506,Z 1152.61,A -85,B 0,C 180,E1 -3062.148,E2 -3062.148} C_VEL
LIN {X 0,Y 20.817,Z 1154.536,A -85,B 0,C 180,E1 -3076.132,E2 -3076.132} C_VEL
LIN {X 0,Y 11.348,Z 1155.008,A -85,B 0,C 180,E1 -3101.454,E2 -3101.454} C_VEL
LIN {X 0,Y 8.364,Z 1155.128,A -85,B 0,C 180,E1 -3115.008,E2 -3115.008} C_VEL
LIN {X 0,Y 3.444,Z 1155.346,A -85,B 0,C 180,E1 -3155.497,E2 -3155.497} C_VEL
LIN {X 0,Y 1.916,Z 1155.412,A -85,B 0,C 180,E1 -3214.583,E2 -3214.583} C_VEL
LIN {X 0,Y 1.364,Z 1155.446,A -85,B 0,C 180,E1 -3236.234,E2 -3236.234} C_VEL
LIN {X 0,Y 1.363,Z 1155.44,A -85,B 0,C 180,E1 -3063.789,E2 -3063.789} C_VEL
LIN {X 0,Y 1.364,Z 1155.446,A -85,B 0,C 180,E1 -3236.234,E2 -3236.234} C_VEL
LIN {X 0,Y 3.381,Z 1157.446,A -85,B 0,C 180,E1 -3243.303,E2 -3243.303} C_VEL
LIN {X 0,Y 3.381,Z 1180,A -85,B 0,C 180,E1 -3243.303,E2 -3243.303} C_VEL
LIN {X 0,Y 3.381,Z 1180,A -85,B 0,C 180,E1 -3243.303,E2 -3243.303}

QRS_NEXT_CUT()

QRS_NEXT()
QRS_HOME()

END
